LIN {X 0,Y 321.804,Z 530.514,A -85,B 0,C 180,E1 -15771.71,E2 -15771.71} C_VEL
LIN {X 0,Y 322.657,Z 517.307,A -85,B 0,C 180,E1 -15772.365,E2 -15772.365} C_VEL
LIN {X 0,Y 323.2,Z 504.38,A -85,B 0,C 180,E1 -15772.747,E2 -15772.747} C_VEL
LIN {X 0,Y 324.606,Z 436.447,A -85,B 0,C 180,E1 -15774.249,E2 -15774.249} C_VEL
LIN {X 0,Y 321.895,Z 423.016,A -85,B 0,C 180,E1 -15774.791,E2 -15774.791} C_VEL
LIN {X 0,Y 315.381,Z 406.695,A -85,B 0,C 180,E1 -15775.746,E2 -15775.746} C_VEL
LIN {X 0,Y 314.625,Z 404.517,A -85,B 0,C 180,E1 -15775.889,E2 -15775.889} C_VEL
LIN {X 0,Y 312.586,Z 395.049,A -85,B 0,C 180,E1 -15779.228,E2 -15779.228} C_VEL
LIN {X 0,Y 312.512,Z 395.055,A -85,B 0,C 180,E1 -15783.492,E2 -15783.492} C_VEL
LIN {X 0,Y 312.529,Z 395.054,A -85,B 0,C 180,E1 -15787.385,E2 -15787.385} C_VEL
LIN {X 0,Y 312.504,Z 395.058,A -85,B 0,C 180,E1 -15789.07,E2 -15789.07} C_VEL
LIN {X 0,Y 311.809,Z 395.146,A -85,B 0,C 180,E1 -15790.146,E2 -15790.146} C_VEL
LIN {X 0,Y 308.949,Z 395.503,A -85,B 0,C 180,E1 -15791.898,E2 -15791.898} C_VEL
LIN {X 0,Y 306.537,Z 395.806,A -85,B 0,C 180,E1 -15793.318,E2 -15793.318} C_VEL
LIN {X 0,Y 305.5,Z 395.932,A -85,B 0,C 180,E1 -15794.418,E2 -15794.418} C_VEL
LIN {X 0,Y 305.412,Z 395.941,A -85,B 0,C 180,E1 -15794.79,E2 -15794.79} C_VEL
LIN {X 0,Y 305.469,Z 395.935,A -85,B 0,C 180,E1 -15798.148,E2 -15798.148} C_VEL
LIN {X 0,Y 305.507,Z 395.922,A -85,B 0,C 180,E1 -15801.602,E2 -15801.602} C_VEL
LIN {X 0,Y 305.467,Z 395.933,A -85,B 0,C 180,E1 -15804.887,E2 -15804.887} C_VEL
LIN {X 0,Y 305.457,Z 395.938,A -85,B 0,C 180,E1 -15808.355,E2 -15808.355} C_VEL
LIN {X 0,Y 305.525,Z 395.924,A -85,B 0,C 180,E1 -15811.114,E2 -15811.114} C_VEL
LIN {X 0,Y 305.576,Z 395.922,A -85,B 0,C 180,E1 -15814.088,E2 -15814.088} C_VEL
LIN {X 0,Y 305.533,Z 395.926,A -85,B 0,C 180,E1 -15818.405,E2 -15818.405} C_VEL
LIN {X 0,Y 305.596,Z 395.913,A -85,B 0,C 180,E1 -15821.218,E2 -15821.218} C_VEL
LIN {X 0,Y 305.653,Z 395.908,A -85,B 0,C 180,E1 -15825.349,E2 -15825.349} C_VEL
LIN {X 0,Y 305.643,Z 395.911,A -85,B 0,C 180,E1 -15829.4,E2 -15829.4} C_VEL
LIN {X 0,Y 305.818,Z 395.887,A -85,B 0,C 180,E1 -15832.074,E2 -15832.074} C_VEL
LIN {X 0,Y 305.694,Z 395.904,A -85,B 0,C 180,E1 -15834.723,E2 -15834.723} C_VEL
LIN {X 0,Y 305.96,Z 395.866,A -85,B 0,C 180,E1 -15838.684,E2 -15838.684} C_VEL
LIN {X 0,Y 305.96,Z 395.871,A -85,B 0,C 180,E1 -15841.316,E2 -15841.316} C_VEL
LIN {X 0,Y 305.69,Z 395.903,A -85,B 0,C 180,E1 -15845.276,E2 -15845.276} C_VEL
LIN {X 0,Y 305.777,Z 395.897,A -85,B 0,C 180,E1 -15847.927,E2 -15847.927} C_VEL
LIN {X 0,Y 305.61,Z 395.915,A -85,B 0,C 180,E1 -15851.945,E2 -15851.945} C_VEL
LIN {X 0,Y 305.642,Z 395.911,A -85,B 0,C 180,E1 -15855.035,E2 -15855.035} C_VEL
LIN {X 0,Y 305.581,Z 395.922,A -85,B 0,C 180,E1 -15859.445,E2 -15859.445} C_VEL
LIN {X 0,Y 305.495,Z 395.927,A -85,B 0,C 180,E1 -15863.041,E2 -15863.041} C_VEL
LIN {X 0,Y 305.535,Z 395.924,A -85,B 0,C 180,E1 -15866.221,E2 -15866.221} C_VEL
LIN {X 0,Y 305.492,Z 395.931,A -85,B 0,C 180,E1 -15869.047,E2 -15869.047} C_VEL
LIN {X 0,Y 305.445,Z 395.935,A -85,B 0,C 180,E1 -15871.952,E2 -15871.952} C_VEL
LIN {X 0,Y 305.466,Z 395.935,A -85,B 0,C 180,E1 -15875.113,E2 -15875.113} C_VEL
LIN {X 0,Y 305.443,Z 395.935,A -85,B 0,C 180,E1 -15878.526,E2 -15878.526} C_VEL
LIN {X 0,Y 305.462,Z 395.934,A -85,B 0,C 180,E1 -15882.586,E2 -15882.586} C_VEL
LIN {X 0,Y 305.445,Z 395.936,A -85,B 0,C 180,E1 -15886.348,E2 -15886.348} C_VEL
LIN {X 0,Y 305.461,Z 395.934,A -85,B 0,C 180,E1 -15889.892,E2 -15889.892} C_VEL
LIN {X 0,Y 305.484,Z 395.933,A -85,B 0,C 180,E1 -15893.631,E2 -15893.631} C_VEL
LIN {X 0,Y 305.546,Z 396.115,A -85,B 0,C 180,E1 -15896.789,E2 -15896.789} C_VEL
LIN {X 0,Y 308.175,Z 407.817,A -85,B 0,C 180,E1 -15900.722,E2 -15900.722} C_VEL
LIN {X 0,Y 310.062,Z 417.52,A -85,B 0,C 180,E1 -15903.763,E2 -15903.763} C_VEL
LIN {X 0,Y 311.791,Z 423.086,A -85,B 0,C 180,E1 -15904.058,E2 -15904.058} C_VEL
LIN {X 0,Y 316.195,Z 447.46,A -85,B 0,C 180,E1 -15905.042,E2 -15905.042} C_VEL
LIN {X 0,Y 317.783,Z 458.385,A -85,B 0,C 180,E1 -15905.441,E2 -15905.441} C_VEL
LIN {X 0,Y 316.113,Z 525.615,A -85,B 0,C 180,E1 -15906.973,E2 -15906.973} C_VEL
LIN {X 0,Y 315.252,Z 538.795,A -85,B 0,C 180,E1 -15907.513,E2 -15907.513} C_VEL
LIN {X 0,Y 314.171,Z 550.908,A -85,B 0,C 180,E1 -15908.253,E2 -15908.253} C_VEL
LIN {X 0,Y 312.715,Z 563.132,A -85,B 0,C 180,E1 -15909.269,E2 -15909.269} C_VEL
LIN {X 0,Y 311.16,Z 574.706,A -85,B 0,C 180,E1 -15910.54,E2 -15910.54} C_VEL
LIN {X 0,Y 309.557,Z 585.128,A -85,B 0,C 180,E1 -15911.981,E2 -15911.981} C_VEL
LIN {X 0,Y 308.213,Z 594.648,A -85,B 0,C 180,E1 -15913.638,E2 -15913.638} C_VEL
LIN {X 0,Y 306.919,Z 602.895,A -85,B 0,C 180,E1 -15915.411,E2 -15915.411} C_VEL
LIN {X 0,Y 305.617,Z 610.319,A -85,B 0,C 180,E1 -15917.381,E2 -15917.381} C_VEL
LIN {X 0,Y 304.721,Z 616.285,A -85,B 0,C 180,E1 -15919.367,E2 -15919.367} C_VEL
LIN {X 0,Y 304.15,Z 621.001,A -85,B 0,C 180,E1 -15921.361,E2 -15921.361} C_VEL
LIN {X 0,Y 303.741,Z 624.604,A -85,B 0,C 180,E1 -15923.356,E2 -15923.356} C_VEL
LIN {X 0,Y 303.618,Z 626.463,A -85,B 0,C 180,E1 -15924.687,E2 -15924.687} C_VEL
LIN {X 0,Y 303.589,Z 627.858,A -85,B 0,C 180,E1 -15926.017,E2 -15926.017} C_VEL
LIN {X 0,Y 303.598,Z 628.855,A -85,B 0,C 180,E1 -15927.346,E2 -15927.346} C_VEL
LIN {X 0,Y 303.556,Z 629.461,A -85,B 0,C 180,E1 -15928.673,E2 -15928.673} C_VEL
LIN {X 0,Y 303.565,Z 629.674,A -85,B 0,C 180,E1 -15930,E2 -15930} C_VEL
LIN {X 0,Y 303.556,Z 629.454,A -85,B 0,C 180,E1 -15931.326,E2 -15931.326} C_VEL
LIN {X 0,Y 303.598,Z 628.844,A -85,B 0,C 180,E1 -15932.653,E2 -15932.653} C_VEL
LIN {X 0,Y 303.589,Z 627.844,A -85,B 0,C 180,E1 -15933.982,E2 -15933.982} C_VEL
LIN {X 0,Y 303.618,Z 626.155,A -85,B 0,C 180,E1 -15935.53,E2 -15935.53} C_VEL
LIN {X 0,Y 303.993,Z 622.272,A -85,B 0,C 180,E1 -15937.973,E2 -15937.973} C_VEL
LIN {X 0,Y 304.49,Z 617.927,A -85,B 0,C 180,E1 -15939.968,E2 -15939.968} C_VEL
LIN {X 0,Y 305.24,Z 612.394,A -85,B 0,C 180,E1 -15941.959,E2 -15941.959} C_VEL
LIN {X 0,Y 306.422,Z 605.493,A -85,B 0,C 180,E1 -15943.935,E2 -15943.935} C_VEL
LIN {X 0,Y 307.55,Z 598.445,A -85,B 0,C 180,E1 -15945.575,E2 -15945.575} C_VEL
LIN {X 0,Y 308.841,Z 589.95,A -85,B 0,C 180,E1 -15947.207,E2 -15947.207} C_VEL
LIN {X 0,Y 310.402,Z 579.455,A -85,B 0,C 180,E1 -15948.823,E2 -15948.823} C_VEL
LIN {X 0,Y 312.114,Z 567.645,A -85,B 0,C 180,E1 -15950.255,E2 -15950.255} C_VEL
LIN {X 0,Y 313.542,Z 555.751,A -85,B 0,C 180,E1 -15951.361,E2 -15951.361} C_VEL
LIN {X 0,Y 314.779,Z 543.373,A -85,B 0,C 180,E1 -15952.22,E2 -15952.22} C_VEL
LIN {X 0,Y 315.807,Z 530.636,A -85,B 0,C 180,E1 -15952.833,E2 -15952.833} C_VEL
LIN {X 0,Y 316.361,Z 517.195,A -85,B 0,C 180,E1 -15953.223,E2 -15953.223} C_VEL
LIN {X 0,Y 317.613,Z 456.986,A -85,B 0,C 180,E1 -15954.583,E2 -15954.583} C_VEL
LIN {X 0,Y 313.2,Z 430.545,A -85,B 0,C 180,E1 -15955.606,E2 -15955.606} C_VEL
LIN {X 0,Y 311.031,Z 420.234,A -85,B 0,C 180,E1 -15956.055,E2 -15956.055} C_VEL
LIN {X 0,Y 309.994,Z 417.236,A -85,B 0,C 180,E1 -15956.25,E2 -15956.25} C_VEL
LIN {X 0,Y 308.239,Z 408.025,A -85,B 0,C 180,E1 -15959.181,E2 -15959.181} C_VEL
LIN {X 0,Y 305.506,Z 395.931,A -85,B 0,C 180,E1 -15963.265,E2 -15963.265} C_VEL
LIN {X 0,Y 305.476,Z 395.934,A -85,B 0,C 180,E1 -15966.739,E2 -15966.739} C_VEL
LIN {X 0,Y 305.455,Z 395.936,A -85,B 0,C 180,E1 -15970.6,E2 -15970.6} C_VEL
LIN {X 0,Y 305.42,Z 395.939,A -85,B 0,C 180,E1 -15974.493,E2 -15974.493} C_VEL
LIN {X 0,Y 305.443,Z 395.935,A -85,B 0,C 180,E1 -15978.143,E2 -15978.143} C_VEL
LIN {X 0,Y 305.468,Z 395.93,A -85,B 0,C 180,E1 -15981.596,E2 -15981.596} C_VEL
LIN {X 0,Y 305.464,Z 395.934,A -85,B 0,C 180,E1 -15984.887,E2 -15984.887} C_VEL
LIN {X 0,Y 305.451,Z 395.936,A -85,B 0,C 180,E1 -15988.356,E2 -15988.356} C_VEL
LIN {X 0,Y 305.514,Z 395.927,A -85,B 0,C 180,E1 -15991.113,E2 -15991.113} C_VEL
LIN {X 0,Y 305.572,Z 395.92,A -85,B 0,C 180,E1 -15994.088,E2 -15994.088} C_VEL
LIN {X 0,Y 305.528,Z 395.928,A -85,B 0,C 180,E1 -15998.405,E2 -15998.405} C_VEL
LIN {X 0,Y 305.592,Z 395.916,A -85,B 0,C 180,E1 -16001.218,E2 -16001.218} C_VEL
LIN {X 0,Y 305.651,Z 395.906,A -85,B 0,C 180,E1 -16005.349,E2 -16005.349} C_VEL
LIN {X 0,Y 305.639,Z 395.909,A -85,B 0,C 180,E1 -16009.4,E2 -16009.4} C_VEL
LIN {X 0,Y 305.774,Z 395.896,A -85,B 0,C 180,E1 -16012.073,E2 -16012.073} C_VEL
LIN {X 0,Y 305.686,Z 395.904,A -85,B 0,C 180,E1 -16014.723,E2 -16014.723} C_VEL
LIN {X 0,Y 305.958,Z 395.872,A -85,B 0,C 180,E1 -16018.684,E2 -16018.684} C_VEL
LIN {X 0,Y 305.96,Z 395.867,A -85,B 0,C 180,E1 -16021.316,E2 -16021.316} C_VEL
LIN {X 0,Y 305.855,Z 395.883,A -85,B 0,C 180,E1 -16026.597,E2 -16026.597} C_VEL
LIN {X 0,Y 305.737,Z 395.899,A -85,B 0,C 180,E1 -16029.26,E2 -16029.26} C_VEL
LIN {X 0,Y 305.591,Z 395.916,A -85,B 0,C 180,E1 -16033.296,E2 -16033.296} C_VEL
LIN {X 0,Y 305.596,Z 395.918,A -85,B 0,C 180,E1 -16036.02,E2 -16036.02} C_VEL
LIN {X 0,Y 305.583,Z 395.919,A -85,B 0,C 180,E1 -16039.447,E2 -16039.447} C_VEL
LIN {X 0,Y 305.493,Z 395.928,A -85,B 0,C 180,E1 -16043.042,E2 -16043.042} C_VEL
LIN {X 0,Y 305.549,Z 395.922,A -85,B 0,C 180,E1 -16046.227,E2 -16046.227} C_VEL
LIN {X 0,Y 305.497,Z 395.929,A -85,B 0,C 180,E1 -16049.05,E2 -16049.05} C_VEL
LIN {X 0,Y 305.447,Z 395.938,A -85,B 0,C 180,E1 -16051.952,E2 -16051.952} C_VEL
LIN {X 0,Y 305.465,Z 395.932,A -85,B 0,C 180,E1 -16055.113,E2 -16055.113} C_VEL
LIN {X 0,Y 305.479,Z 395.93,A -85,B 0,C 180,E1 -16058.536,E2 -16058.536} C_VEL
LIN {X 0,Y 305.476,Z 395.931,A -85,B 0,C 180,E1 -16062.59,E2 -16062.59} C_VEL
LIN {X 0,Y 305.456,Z 395.936,A -85,B 0,C 180,E1 -16067.414,E2 -16067.414} C_VEL
LIN {X 0,Y 305.478,Z 395.934,A -85,B 0,C 180,E1 -16071.598,E2 -16071.598} C_VEL
LIN {X 0,Y 305.464,Z 395.935,A -85,B 0,C 180,E1 -16074.887,E2 -16074.887} C_VEL
LIN {X 0,Y 305.454,Z 395.937,A -85,B 0,C 180,E1 -16078.355,E2 -16078.355} C_VEL
LIN {X 0,Y 305.519,Z 395.981,A -85,B 0,C 180,E1 -16080.42,E2 -16080.42} C_VEL
LIN {X 0,Y 307.484,Z 404.768,A -85,B 0,C 180,E1 -16083.603,E2 -16083.603} C_VEL
LIN {X 0,Y 315.927,Z 426.072,A -85,B 0,C 180,E1 -16084.895,E2 -16084.895} C_VEL
LIN {X 0,Y 318.22,Z 437.996,A -85,B 0,C 180,E1 -16085.381,E2 -16085.381} C_VEL
LIN {X 0,Y 316.423,Z 511.235,A -85,B 0,C 180,E1 -16087.041,E2 -16087.041} C_VEL
LIN {X 0,Y 315.6,Z 524.625,A -85,B 0,C 180,E1 -16087.583,E2 -16087.583} C_VEL
LIN {X 0,Y 314.558,Z 537.389,A -85,B 0,C 180,E1 -16088.368,E2 -16088.368} C_VEL
LIN {X 0,Y 313.347,Z 548.722,A -85,B 0,C 180,E1 -16089.314,E2 -16089.314} C_VEL
LIN {X 0,Y 311.903,Z 560.369,A -85,B 0,C 180,E1 -16090.588,E2 -16090.588} C_VEL
LIN {X 0,Y 310.383,Z 571.362,A -85,B 0,C 180,E1 -16092.117,E2 -16092.117} C_VEL
LIN {X 0,Y 308.925,Z 581.06,A -85,B 0,C 180,E1 -16093.818,E2 -16093.818} C_VEL
LIN {X 0,Y 307.357,Z 589.977,A -85,B 0,C 180,E1 -16095.771,E2 -16095.771} C_VEL
LIN {X 0,Y 306.173,Z 597.152,A -85,B 0,C 180,E1 -16097.741,E2 -16097.741} C_VEL
LIN {X 0,Y 305.366,Z 601.99,A -85,B 0,C 180,E1 -16099.39,E2 -16099.39} C_VEL
LIN {X 0,Y 304.611,Z 606.691,A -85,B 0,C 180,E1 -16101.375,E2 -16101.375} C_VEL
LIN {X 0,Y 304.105,Z 610.649,A -85,B 0,C 180,E1 -16103.593,E2 -16103.593} C_VEL
LIN {X 0,Y 303.82,Z 613.541,A -85,B 0,C 180,E1 -16106.021,E2 -16106.021} C_VEL
LIN {X 0,Y 303.598,Z 615.148,A -85,B 0,C 180,E1 -16108.674,E2 -16108.674} C_VEL
LIN {X 0,Y 303.571,Z 615.38,A -85,B 0,C 180,E1 -16110,E2 -16110} C_VEL
LIN {X 0,Y 303.598,Z 615.187,A -85,B 0,C 180,E1 -16111.327,E2 -16111.327} C_VEL
LIN {X 0,Y 303.817,Z 613.631,A -85,B 0,C 180,E1 -16113.98,E2 -16113.98} C_VEL
LIN {X 0,Y 304.071,Z 610.898,A -85,B 0,C 180,E1 -16116.35,E2 -16116.35} C_VEL
LIN {X 0,Y 304.609,Z 606.928,A -85,B 0,C 180,E1 -16118.625,E2 -16118.625} C_VEL
LIN {X 0,Y 305.318,Z 602.291,A -85,B 0,C 180,E1 -16120.612,E2 -16120.612} C_VEL
LIN {X 0,Y 306.51,Z 595.298,A -85,B 0,C 180,E1 -16122.918,E2 -16122.918} C_VEL
LIN {X 0,Y 307.787,Z 587.719,A -85,B 0,C 180,E1 -16124.885,E2 -16124.885} C_VEL
LIN {X 0,Y 309.433,Z 578.177,A -85,B 0,C 180,E1 -16126.833,E2 -16126.833} C_VEL
LIN {X 0,Y 310.835,Z 568.331,A -85,B 0,C 180,E1 -16128.454,E2 -16128.454} C_VEL
LIN {X 0,Y 312.169,Z 558.637,A -85,B 0,C 180,E1 -16129.737,E2 -16129.737} C_VEL
LIN {X 0,Y 313.521,Z 548.137,A -85,B 0,C 180,E1 -16130.847,E2 -16130.847} C_VEL
LIN {X 0,Y 314.84,Z 535.491,A -85,B 0,C 180,E1 -16131.871,E2 -16131.871} C_VEL
LIN {X 0,Y 315.792,Z 522.821,A -85,B 0,C 180,E1 -16132.619,E2 -16132.619} C_VEL
LIN {X 0,Y 316.469,Z 510.728,A -85,B 0,C 180,E1 -16133.086,E2 -16133.086} C_VEL
LIN {X 0,Y 318.156,Z 437.661,A -85,B 0,C 180,E1 -16134.747,E2 -16134.747} C_VEL
LIN {X 0,Y 315.68,Z 425.321,A -85,B 0,C 180,E1 -16135.26,E2 -16135.26} C_VEL
LIN {X 0,Y 308.519,Z 407.482,A -85,B 0,C 180,E1 -16136.346,E2 -16136.346} C_VEL
LIN {X 0,Y 307.462,Z 404.709,A -85,B 0,C 180,E1 -16136.533,E2 -16136.533} C_VEL
LIN {X 0,Y 305.524,Z 395.929,A -85,B 0,C 180,E1 -16139.776,E2 -16139.776} C_VEL
LIN {X 0,Y 305.468,Z 395.934,A -85,B 0,C 180,E1 -16144.079,E2 -16144.079} C_VEL
LIN {X 0,Y 305.478,Z 395.932,A -85,B 0,C 180,E1 -16146.74,E2 -16146.74} C_VEL
LIN {X 0,Y 305.458,Z 395.937,A -85,B 0,C 180,E1 -16150.6,E2 -16150.6} C_VEL
LIN {X 0,Y 305.422,Z 395.942,A -85,B 0,C 180,E1 -16154.493,E2 -16154.493} C_VEL
LIN {X 0,Y 305.412,Z 395.941,A -85,B 0,C 180,E1 -16154.79,E2 -16154.79} C_VEL
LIN {X 0,Y 304.74,Z 396.024,A -85,B 0,C 180,E1 -16155.891,E2 -16155.891} C_VEL
LIN {X 0,Y 301.904,Z 396.377,A -85,B 0,C 180,E1 -16157.684,E2 -16157.684} C_VEL
LIN {X 0,Y 299.511,Z 396.67,A -85,B 0,C 180,E1 -16159.138,E2 -16159.138} C_VEL
LIN {X 0,Y 298.494,Z 396.795,A -85,B 0,C 180,E1 -16160.264,E2 -16160.264} C_VEL
LIN {X 0,Y 298.417,Z 396.804,A -85,B 0,C 180,E1 -16160.645,E2 -16160.645} C_VEL
LIN {X 0,Y 298.436,Z 396.809,A -85,B 0,C 180,E1 -16163.932,E2 -16163.932} C_VEL
LIN {X 0,Y 298.4,Z 396.815,A -85,B 0,C 180,E1 -16167.983,E2 -16167.983} C_VEL
LIN {X 0,Y 298.468,Z 396.805,A -85,B 0,C 180,E1 -16171.905,E2 -16171.905} C_VEL
LIN {X 0,Y 298.49,Z 396.798,A -85,B 0,C 180,E1 -16174.924,E2 -16174.924} C_VEL
LIN {X 0,Y 298.469,Z 396.803,A -85,B 0,C 180,E1 -16179.317,E2 -16179.317} C_VEL
LIN {X 0,Y 298.543,Z 396.797,A -85,B 0,C 180,E1 -16182.18,E2 -16182.18} C_VEL
LIN {X 0,Y 298.598,Z 396.787,A -85,B 0,C 180,E1 -16184.995,E2 -16184.995} C_VEL
LIN {X 0,Y 298.598,Z 396.788,A -85,B 0,C 180,E1 -16189.147,E2 -16189.147} C_VEL
LIN {X 0,Y 298.763,Z 396.767,A -85,B 0,C 180,E1 -16191.886,E2 -16191.886} C_VEL
LIN {X 0,Y 298.665,Z 396.78,A -85,B 0,C 180,E1 -16194.599,E2 -16194.599} C_VEL
LIN {X 0,Y 298.927,Z 396.742,A -85,B 0,C 180,E1 -16198.653,E2 -16198.653} C_VEL
LIN {X 0,Y 298.927,Z 396.747,A -85,B 0,C 180,E1 -16201.347,E2 -16201.347} C_VEL
LIN {X 0,Y 298.782,Z 396.763,A -85,B 0,C 180,E1 -16206.754,E2 -16206.754} C_VEL
LIN {X 0,Y 298.636,Z 396.787,A -85,B 0,C 180,E1 -16209.482,E2 -16209.482} C_VEL
LIN {X 0,Y 298.558,Z 396.796,A -85,B 0,C 180,E1 -16213.615,E2 -16213.615} C_VEL
LIN {X 0,Y 298.553,Z 396.791,A -85,B 0,C 180,E1 -16216.408,E2 -16216.408} C_VEL
LIN {X 0,Y 298.516,Z 396.802,A -85,B 0,C 180,E1 -16219.655,E2 -16219.655} C_VEL
LIN {X 0,Y 298.461,Z 396.808,A -85,B 0,C 180,E1 -16223.597,E2 -16223.597} C_VEL
LIN {X 0,Y 298.49,Z 396.801,A -85,B 0,C 180,E1 -16226.574,E2 -16226.574} C_VEL
LIN {X 0,Y 298.42,Z 396.812,A -85,B 0,C 180,E1 -16229.641,E2 -16229.641} C_VEL
LIN {X 0,Y 298.398,Z 396.813,A -85,B 0,C 180,E1 -16232.8,E2 -16232.8} C_VEL
LIN {X 0,Y 298.447,Z 396.808,A -85,B 0,C 180,E1 -16236.807,E2 -16236.807} C_VEL
LIN {X 0,Y 298.391,Z 396.818,A -85,B 0,C 180,E1 -16241.088,E2 -16241.088} C_VEL
LIN {X 0,Y 298.391,Z 396.818,A -85,B 0,C 180,E1 -16245.041,E2 -16245.041} C_VEL
LIN {X 0,Y 298.391,Z 396.818,A -85,B 0,C 180,E1 -16248.912,E2 -16248.912} C_VEL
LIN {X 0,Y 298.449,Z 396.81,A -85,B 0,C 180,E1 -16253.192,E2 -16253.192} C_VEL
LIN {X 0,Y 298.451,Z 396.866,A -85,B 0,C 180,E1 -16256.197,E2 -16256.197} C_VEL
LIN {X 0,Y 300.988,Z 407.974,A -85,B 0,C 180,E1 -16260.058,E2 -16260.058} C_VEL
LIN {X 0,Y 302.821,Z 417.308,A -85,B 0,C 180,E1 -16263.085,E2 -16263.085} C_VEL
LIN {X 0,Y 305.502,Z 424.753,A -85,B 0,C 180,E1 -16263.53,E2 -16263.53} C_VEL
LIN {X 0,Y 309.917,Z 449.444,A -85,B 0,C 180,E1 -16264.554,E2 -16264.554} C_VEL
LIN {X 0,Y 311.305,Z 459.53,A -85,B 0,C 180,E1 -16264.927,E2 -16264.927} C_VEL
LIN {X 0,Y 309.595,Z 525.461,A -85,B 0,C 180,E1 -16266.46,E2 -16266.46} C_VEL
LIN {X 0,Y 308.704,Z 538.637,A -85,B 0,C 180,E1 -16267.009,E2 -16267.009} C_VEL
LIN {X 0,Y 307.593,Z 550.747,A -85,B 0,C 180,E1 -16267.763,E2 -16267.763} C_VEL
LIN {X 0,Y 306.089,Z 562.97,A -85,B 0,C 180,E1 -16268.799,E2 -16268.799} C_VEL
LIN {X 0,Y 304.483,Z 574.543,A -85,B 0,C 180,E1 -16270.095,E2 -16270.095} C_VEL
LIN {X 0,Y 302.773,Z 584.963,A -85,B 0,C 180,E1 -16271.562,E2 -16271.562} C_VEL
LIN {X 0,Y 301.516,Z 593.488,A -85,B 0,C 180,E1 -16273.06,E2 -16273.06} C_VEL
LIN {X 0,Y 300.281,Z 601.354,A -85,B 0,C 180,E1 -16274.733,E2 -16274.733} C_VEL
LIN {X 0,Y 298.857,Z 609.032,A -85,B 0,C 180,E1 -16276.745,E2 -16276.745} C_VEL
LIN {X 0,Y 297.727,Z 616.119,A -85,B 0,C 180,E1 -16279.114,E2 -16279.114} C_VEL
LIN {X 0,Y 297.092,Z 620.834,A -85,B 0,C 180,E1 -16281.155,E2 -16281.155} C_VEL
LIN {X 0,Y 296.688,Z 624.438,A -85,B 0,C 180,E1 -16283.198,E2 -16283.198} C_VEL
LIN {X 0,Y 296.532,Z 626.296,A -85,B 0,C 180,E1 -16284.56,E2 -16284.56} C_VEL
LIN {X 0,Y 296.49,Z 627.691,A -85,B 0,C 180,E1 -16285.922,E2 -16285.922} C_VEL
LIN {X 0,Y 296.523,Z 628.688,A -85,B 0,C 180,E1 -16287.283,E2 -16287.283} C_VEL
LIN {X 0,Y 296.476,Z 629.294,A -85,B 0,C 180,E1 -16288.641,E2 -16288.641} C_VEL
LIN {X 0,Y 296.482,Z 629.508,A -85,B 0,C 180,E1 -16290,E2 -16290} C_VEL
LIN {X 0,Y 296.476,Z 629.287,A -85,B 0,C 180,E1 -16291.358,E2 -16291.358} C_VEL
LIN {X 0,Y 296.523,Z 628.677,A -85,B 0,C 180,E1 -16292.717,E2 -16292.717} C_VEL
LIN {X 0,Y 296.49,Z 627.677,A -85,B 0,C 180,E1 -16294.078,E2 -16294.078} C_VEL
LIN {X 0,Y 296.546,Z 626.189,A -85,B 0,C 180,E1 -16295.508,E2 -16295.508} C_VEL
LIN {X 0,Y 296.796,Z 623.333,A -85,B 0,C 180,E1 -16297.483,E2 -16297.483} C_VEL
LIN {X 0,Y 297.274,Z 619.354,A -85,B 0,C 180,E1 -16299.526,E2 -16299.526} C_VEL
LIN {X 0,Y 298.128,Z 613.237,A -85,B 0,C 180,E1 -16301.904,E2 -16301.904} C_VEL
LIN {X 0,Y 299.301,Z 606.56,A -85,B 0,C 180,E1 -16303.927,E2 -16303.927} C_VEL
LIN {X 0,Y 300.683,Z 598.275,A -85,B 0,C 180,E1 -16305.94,E2 -16305.94} C_VEL
LIN {X 0,Y 302.043,Z 589.78,A -85,B 0,C 180,E1 -16307.607,E2 -16307.607} C_VEL
LIN {X 0,Y 303.666,Z 579.284,A -85,B 0,C 180,E1 -16309.256,E2 -16309.256} C_VEL
LIN {X 0,Y 305.454,Z 567.473,A -85,B 0,C 180,E1 -16310.717,E2 -16310.717} C_VEL
LIN {X 0,Y 306.952,Z 555.579,A -85,B 0,C 180,E1 -16311.843,E2 -16311.843} C_VEL
LIN {X 0,Y 308.219,Z 543.198,A -85,B 0,C 180,E1 -16312.719,E2 -16312.719} C_VEL
LIN {X 0,Y 309.285,Z 530.458,A -85,B 0,C 180,E1 -16313.343,E2 -16313.343} C_VEL
LIN {X 0,Y 309.851,Z 517.007,A -85,B 0,C 180,E1 -16313.741,E2 -16313.741} C_VEL
LIN {X 0,Y 311.196,Z 458.096,A -85,B 0,C 180,E1 -16315.093,E2 -16315.093} C_VEL
LIN {X 0,Y 306.801,Z 431.766,A -85,B 0,C 180,E1 -16316.144,E2 -16316.144} C_VEL
LIN {X 0,Y 304.983,Z 422.969,A -85,B 0,C 180,E1 -16316.537,E2 -16316.537} C_VEL
LIN {X 0,Y 302.765,Z 417.024,A -85,B 0,C 180,E1 -16316.935,E2 -16316.935} C_VEL
LIN {X 0,Y 300.809,Z 407.187,A -85,B 0,C 180,E1 -16320.179,E2 -16320.179} C_VEL
LIN {X 0,Y 298.45,Z 396.81,A -85,B 0,C 180,E1 -16323.802,E2 -16323.802} C_VEL
LIN {X 0,Y 298.415,Z 396.812,A -85,B 0,C 180,E1 -16327.758,E2 -16327.758} C_VEL
LIN {X 0,Y 298.386,Z 396.816,A -85,B 0,C 180,E1 -16331.261,E2 -16331.261} C_VEL
LIN {X 0,Y 298.389,Z 396.818,A -85,B 0,C 180,E1 -16335.041,E2 -16335.041} C_VEL
LIN {X 0,Y 298.389,Z 396.815,A -85,B 0,C 180,E1 -16338.912,E2 -16338.912} C_VEL
LIN {X 0,Y 298.445,Z 396.808,A -85,B 0,C 180,E1 -16343.193,E2 -16343.193} C_VEL
LIN {X 0,Y 298.396,Z 396.814,A -85,B 0,C 180,E1 -16347.2,E2 -16347.2} C_VEL
LIN {X 0,Y 298.428,Z 396.813,A -85,B 0,C 180,E1 -16350.616,E2 -16350.616} C_VEL
LIN {X 0,Y 298.479,Z 396.803,A -85,B 0,C 180,E1 -16353.476,E2 -16353.476} C_VEL
LIN {X 0,Y 298.437,Z 396.81,A -85,B 0,C 180,E1 -16356.697,E2 -16356.697} C_VEL
LIN {X 0,Y 298.541,Z 396.796,A -85,B 0,C 180,E1 -16360.757,E2 -16360.757} C_VEL
LIN {X 0,Y 298.595,Z 396.786,A -85,B 0,C 180,E1 -16364.995,E2 -16364.995} C_VEL
LIN {X 0,Y 298.595,Z 396.787,A -85,B 0,C 180,E1 -16369.147,E2 -16369.147} C_VEL
LIN {X 0,Y 298.72,Z 396.773,A -85,B 0,C 180,E1 -16371.885,E2 -16371.885} C_VEL
LIN {X 0,Y 298.657,Z 396.78,A -85,B 0,C 180,E1 -16374.599,E2 -16374.599} C_VEL
LIN {X 0,Y 298.924,Z 396.749,A -85,B 0,C 180,E1 -16378.653,E2 -16378.653} C_VEL
LIN {X 0,Y 298.926,Z 396.743,A -85,B 0,C 180,E1 -16381.347,E2 -16381.347} C_VEL
LIN {X 0,Y 298.8,Z 396.761,A -85,B 0,C 180,E1 -16386.754,E2 -16386.754} C_VEL
LIN {X 0,Y 298.682,Z 396.778,A -85,B 0,C 180,E1 -16389.481,E2 -16389.481} C_VEL
LIN {X 0,Y 298.554,Z 396.794,A -85,B 0,C 180,E1 -16393.615,E2 -16393.615} C_VEL
LIN {X 0,Y 298.551,Z 396.792,A -85,B 0,C 180,E1 -16396.409,E2 -16396.409} C_VEL
LIN {X 0,Y 298.518,Z 396.801,A -85,B 0,C 180,E1 -16399.657,E2 -16399.657} C_VEL
LIN {X 0,Y 298.459,Z 396.807,A -85,B 0,C 180,E1 -16403.598,E2 -16403.598} C_VEL
LIN {X 0,Y 298.491,Z 396.8,A -85,B 0,C 180,E1 -16406.574,E2 -16406.574} C_VEL
LIN {X 0,Y 298.422,Z 396.813,A -85,B 0,C 180,E1 -16409.641,E2 -16409.641} C_VEL
LIN {X 0,Y 298.398,Z 396.813,A -85,B 0,C 180,E1 -16412.8,E2 -16412.8} C_VEL
LIN {X 0,Y 298.467,Z 396.804,A -85,B 0,C 180,E1 -16416.813,E2 -16416.813} C_VEL
LIN {X 0,Y 298.415,Z 396.811,A -85,B 0,C 180,E1 -16421.094,E2 -16421.094} C_VEL
LIN {X 0,Y 298.355,Z 396.819,A -85,B 0,C 180,E1 -16425.035,E2 -16425.035} C_VEL
LIN {X 0,Y 298.386,Z 396.816,A -85,B 0,C 180,E1 -16428.739,E2 -16428.739} C_VEL
LIN {X 0,Y 298.416,Z 396.812,A -85,B 0,C 180,E1 -16432.242,E2 -16432.242} C_VEL
LIN {X 0,Y 298.41,Z 396.814,A -85,B 0,C 180,E1 -16435.581,E2 -16435.581} C_VEL
LIN {X 0,Y 298.468,Z 396.936,A -85,B 0,C 180,E1 -16439.927,E2 -16439.927} C_VEL
LIN {X 0,Y 300.277,Z 404.892,A -85,B 0,C 180,E1 -16442.896,E2 -16442.896} C_VEL
LIN {X 0,Y 308.044,Z 423.883,A -85,B 0,C 180,E1 -16444.144,E2 -16444.144} C_VEL
LIN {X 0,Y 310.011,Z 429.691,A -85,B 0,C 180,E1 -16444.468,E2 -16444.468} C_VEL
LIN {X 0,Y 311.75,Z 439.041,A -85,B 0,C 180,E1 -16444.856,E2 -16444.856} C_VEL
LIN {X 0,Y 309.917,Z 511.419,A -85,B 0,C 180,E1 -16446.53,E2 -16446.53} C_VEL
LIN {X 0,Y 309.071,Z 524.802,A -85,B 0,C 180,E1 -16447.082,E2 -16447.082} C_VEL
LIN {X 0,Y 307.986,Z 537.563,A -85,B 0,C 180,E1 -16447.882,E2 -16447.882} C_VEL
LIN {X 0,Y 306.731,Z 548.894,A -85,B 0,C 180,E1 -16448.846,E2 -16448.846} C_VEL
LIN {X 0,Y 305.216,Z 560.54,A -85,B 0,C 180,E1 -16450.145,E2 -16450.145} C_VEL
LIN {X 0,Y 303.81,Z 570.356,A -85,B 0,C 180,E1 -16451.523,E2 -16451.523} C_VEL
LIN {X 0,Y 302.431,Z 579.537,A -85,B 0,C 180,E1 -16453.113,E2 -16453.113} C_VEL
LIN {X 0,Y 301.009,Z 587.409,A -85,B 0,C 180,E1 -16454.772,E2 -16454.772} C_VEL
LIN {X 0,Y 299.647,Z 595.099,A -85,B 0,C 180,E1 -16456.781,E2 -16456.781} C_VEL
LIN {X 0,Y 298.385,Z 602.159,A -85,B 0,C 180,E1 -16459.139,E2 -16459.139} C_VEL
LIN {X 0,Y 297.592,Z 606.86,A -85,B 0,C 180,E1 -16461.17,E2 -16461.17} C_VEL
LIN {X 0,Y 297.024,Z 611.062,A -85,B 0,C 180,E1 -16463.608,E2 -16463.608} C_VEL
LIN {X 0,Y 296.738,Z 613.709,A -85,B 0,C 180,E1 -16465.926,E2 -16465.926} C_VEL
LIN {X 0,Y 296.61,Z 614.703,A -85,B 0,C 180,E1 -16467.284,E2 -16467.284} C_VEL
LIN {X 0,Y 296.488,Z 615.546,A -85,B 0,C 180,E1 -16470,E2 -16470} C_VEL
LIN {X 0,Y 296.518,Z 615.354,A -85,B 0,C 180,E1 -16471.358,E2 -16471.358} C_VEL
LIN {X 0,Y 296.609,Z 614.767,A -85,B 0,C 180,E1 -16472.716,E2 -16472.716} C_VEL
LIN {X 0,Y 296.736,Z 613.798,A -85,B 0,C 180,E1 -16474.075,E2 -16474.075} C_VEL
LIN {X 0,Y 296.997,Z 611.27,A -85,B 0,C 180,E1 -16476.345,E2 -16476.345} C_VEL
LIN {X 0,Y 297.59,Z 607.094,A -85,B 0,C 180,E1 -16478.831,E2 -16478.831} C_VEL
LIN {X 0,Y 298.341,Z 602.456,A -85,B 0,C 180,E1 -16480.863,E2 -16480.863} C_VEL
LIN {X 0,Y 299.557,Z 595.464,A -85,B 0,C 180,E1 -16483.224,E2 -16483.224} C_VEL
LIN {X 0,Y 300.94,Z 587.884,A -85,B 0,C 180,E1 -16485.232,E2 -16485.232} C_VEL
LIN {X 0,Y 302.638,Z 578.341,A -85,B 0,C 180,E1 -16487.223,E2 -16487.223} C_VEL
LIN {X 0,Y 304.094,Z 568.494,A -85,B 0,C 180,E1 -16488.879,E2 -16488.879} C_VEL
LIN {X 0,Y 305.506,Z 558.799,A -85,B 0,C 180,E1 -16490.186,E2 -16490.186} C_VEL
LIN {X 0,Y 306.91,Z 548.298,A -85,B 0,C 180,E1 -16491.317,E2 -16491.317} C_VEL
LIN {X 0,Y 308.255,Z 535.65,A -85,B 0,C 180,E1 -16492.363,E2 -16492.363} C_VEL
LIN {X 0,Y 309.267,Z 522.977,A -85,B 0,C 180,E1 -16493.124,E2 -16493.124} C_VEL
LIN {X 0,Y 309.969,Z 510.875,A -85,B 0,C 180,E1 -16493.599,E2 -16493.599} C_VEL
LIN {X 0,Y 311.742,Z 438.654,A -85,B 0,C 180,E1 -16495.27,E2 -16495.27} C_VEL
LIN {X 0,Y 309.528,Z 427.798,A -85,B 0,C 180,E1 -16495.739,E2 -16495.739} C_VEL
LIN {X 0,Y 302.552,Z 410.393,A -85,B 0,C 180,E1 -16496.835,E2 -16496.835} C_VEL
LIN {X 0,Y 300.286,Z 404.93,A -85,B 0,C 180,E1 -16497.206,E2 -16497.206} C_VEL
LIN {X 0,Y 298.451,Z 396.81,A -85,B 0,C 180,E1 -16500.32,E2 -16500.32} C_VEL
LIN {X 0,Y 298.431,Z 396.814,A -85,B 0,C 180,E1 -16504.488,E2 -16504.488} C_VEL
LIN {X 0,Y 298.417,Z 396.812,A -85,B 0,C 180,E1 -16507.758,E2 -16507.758} C_VEL
LIN {X 0,Y 298.388,Z 396.815,A -85,B 0,C 180,E1 -16511.262,E2 -16511.262} C_VEL
LIN {X 0,Y 298.391,Z 396.814,A -85,B 0,C 180,E1 -16515.042,E2 -16515.042} C_VEL
LIN {X 0,Y 298.417,Z 396.809,A -85,B 0,C 180,E1 -16518.744,E2 -16518.744} C_VEL
LIN {X 0,Y 298.417,Z 396.804,A -85,B 0,C 180,E1 -16520.645,E2 -16520.645} C_VEL
LIN {X 0,Y 297.763,Z 396.888,A -85,B 0,C 180,E1 -16521.772,E2 -16521.772} C_VEL
LIN {X 0,Y 294.914,Z 397.249,A -85,B 0,C 180,E1 -16523.607,E2 -16523.607} C_VEL
LIN {X 0,Y 292.481,Z 397.552,A -85,B 0,C 180,E1 -16525.096,E2 -16525.096} C_VEL
LIN {X 0,Y 291.426,Z 397.682,A -85,B 0,C 180,E1 -16526.249,E2 -16526.249} C_VEL
LIN {X 0,Y 291.334,Z 397.692,A -85,B 0,C 180,E1 -16526.64,E2 -16526.64} C_VEL
LIN {X 0,Y 291.391,Z 397.686,A -85,B 0,C 180,E1 -16530.26,E2 -16530.26} C_VEL
LIN {X 0,Y 291.421,Z 397.682,A -85,B 0,C 180,E1 -16534.272,E2 -16534.272} C_VEL
LIN {X 0,Y 291.394,Z 397.685,A -85,B 0,C 180,E1 -16537.3,E2 -16537.3} C_VEL
LIN {X 0,Y 291.468,Z 397.675,A -85,B 0,C 180,E1 -16540.271,E2 -16540.271} C_VEL
LIN {X 0,Y 291.559,Z 397.664,A -85,B 0,C 180,E1 -16544.624,E2 -16544.624} C_VEL
LIN {X 0,Y 291.541,Z 397.667,A -85,B 0,C 180,E1 -16548.881,E2 -16548.881} C_VEL
LIN {X 0,Y 291.714,Z 397.647,A -85,B 0,C 180,E1 -16551.689,E2 -16551.689} C_VEL
LIN {X 0,Y 291.636,Z 397.656,A -85,B 0,C 180,E1 -16554.468,E2 -16554.468} C_VEL
LIN {X 0,Y 291.893,Z 397.618,A -85,B 0,C 180,E1 -16558.62,E2 -16558.62} C_VEL
LIN {X 0,Y 291.893,Z 397.623,A -85,B 0,C 180,E1 -16561.38,E2 -16561.38} C_VEL
LIN {X 0,Y 291.729,Z 397.641,A -85,B 0,C 180,E1 -16566.918,E2 -16566.918} C_VEL
LIN {X 0,Y 291.577,Z 397.665,A -85,B 0,C 180,E1 -16569.714,E2 -16569.714} C_VEL
LIN {X 0,Y 291.527,Z 397.671,A -85,B 0,C 180,E1 -16573.95,E2 -16573.95} C_VEL
LIN {X 0,Y 291.491,Z 397.67,A -85,B 0,C 180,E1 -16576.818,E2 -16576.818} C_VEL
LIN {X 0,Y 291.454,Z 397.68,A -85,B 0,C 180,E1 -16579.875,E2 -16579.875} C_VEL
LIN {X 0,Y 291.404,Z 397.685,A -85,B 0,C 180,E1 -16584.205,E2 -16584.205} C_VEL
LIN {X 0,Y 291.423,Z 397.686,A -85,B 0,C 180,E1 -16587.271,E2 -16587.271} C_VEL
LIN {X 0,Y 291.338,Z 397.691,A -85,B 0,C 180,E1 -16590.437,E2 -16590.437} C_VEL
LIN {X 0,Y 291.348,Z 397.692,A -85,B 0,C 180,E1 -16593.698,E2 -16593.698} C_VEL
LIN {X 0,Y 291.376,Z 397.691,A -85,B 0,C 180,E1 -16597.253,E2 -16597.253} C_VEL
LIN {X 0,Y 291.336,Z 397.693,A -85,B 0,C 180,E1 -16600.642,E2 -16600.642} C_VEL
LIN {X 0,Y 291.316,Z 397.696,A -85,B 0,C 180,E1 -16604.397,E2 -16604.397} C_VEL
LIN {X 0,Y 291.33,Z 397.696,A -85,B 0,C 180,E1 -16608.404,E2 -16608.404} C_VEL
LIN {X 0,Y 291.356,Z 397.694,A -85,B 0,C 180,E1 -16611.158,E2 -16611.158} C_VEL
LIN {X 0,Y 291.364,Z 397.691,A -85,B 0,C 180,E1 -16614.626,E2 -16614.626} C_VEL
LIN {X 0,Y 291.407,Z 397.83,A -85,B 0,C 180,E1 -16615.654,E2 -16615.654} C_VEL
LIN {X 0,Y 293.836,Z 408.359,A -85,B 0,C 180,E1 -16619.435,E2 -16619.435} C_VEL
LIN {X 0,Y 295.6,Z 417.085,A -85,B 0,C 180,E1 -16622.371,E2 -16622.371} C_VEL
LIN {X 0,Y 299.436,Z 427.211,A -85,B 0,C 180,E1 -16623.019,E2 -16623.019} C_VEL
LIN {X 0,Y 304.085,Z 454.057,A -85,B 0,C 180,E1 -16624.152,E2 -16624.152} C_VEL
LIN {X 0,Y 304.842,Z 460.604,A -85,B 0,C 180,E1 -16624.388,E2 -16624.388} C_VEL
LIN {X 0,Y 303.08,Z 525.307,A -85,B 0,C 180,E1 -16625.922,E2 -16625.922} C_VEL
LIN {X 0,Y 302.128,Z 539.241,A -85,B 0,C 180,E1 -16626.524,E2 -16626.524} C_VEL
LIN {X 0,Y 300.885,Z 551.699,A -85,B 0,C 180,E1 -16627.331,E2 -16627.331} C_VEL
LIN {X 0,Y 299.491,Z 562.808,A -85,B 0,C 180,E1 -16628.309,E2 -16628.309} C_VEL
LIN {X 0,Y 297.823,Z 574.38,A -85,B 0,C 180,E1 -16629.63,E2 -16629.63} C_VEL
LIN {X 0,Y 296.053,Z 584.799,A -85,B 0,C 180,E1 -16631.128,E2 -16631.128} C_VEL
LIN {X 0,Y 294.581,Z 594.049,A -85,B 0,C 180,E1 -16632.799,E2 -16632.799} C_VEL
LIN {X 0,Y 293.128,Z 602.563,A -85,B 0,C 180,E1 -16634.708,E2 -16634.708} C_VEL
LIN {X 0,Y 291.703,Z 609.986,A -85,B 0,C 180,E1 -16636.768,E2 -16636.768} C_VEL
LIN {X 0,Y 290.743,Z 615.952,A -85,B 0,C 180,E1 -16638.85,E2 -16638.85} C_VEL
LIN {X 0,Y 290.054,Z 620.667,A -85,B 0,C 180,E1 -16640.938,E2 -16640.938} C_VEL
LIN {X 0,Y 289.608,Z 624.271,A -85,B 0,C 180,E1 -16643.03,E2 -16643.03} C_VEL
LIN {X 0,Y 289.428,Z 626.328,A -85,B 0,C 180,E1 -16644.612,E2 -16644.612} C_VEL
LIN {X 0,Y 289.427,Z 628.521,A -85,B 0,C 180,E1 -16647.216,E2 -16647.216} C_VEL
LIN {X 0,Y 289.399,Z 629.128,A -85,B 0,C 180,E1 -16648.608,E2 -16648.608} C_VEL
LIN {X 0,Y 289.401,Z 629.341,A -85,B 0,C 180,E1 -16650,E2 -16650} C_VEL
LIN {X 0,Y 289.398,Z 629.12,A -85,B 0,C 180,E1 -16651.391,E2 -16651.391} C_VEL
LIN {X 0,Y 289.427,Z 628.51,A -85,B 0,C 180,E1 -16652.783,E2 -16652.783} C_VEL
LIN {X 0,Y 289.477,Z 626.107,A -85,B 0,C 180,E1 -16655.573,E2 -16655.573} C_VEL
LIN {X 0,Y 289.729,Z 623.164,A -85,B 0,C 180,E1 -16657.667,E2 -16657.667} C_VEL
LIN {X 0,Y 290.255,Z 619.185,A -85,B 0,C 180,E1 -16659.758,E2 -16659.758} C_VEL
LIN {X 0,Y 291.132,Z 613.067,A -85,B 0,C 180,E1 -16662.194,E2 -16662.194} C_VEL
LIN {X 0,Y 292.375,Z 606.39,A -85,B 0,C 180,E1 -16664.264,E2 -16664.264} C_VEL
LIN {X 0,Y 293.843,Z 598.105,A -85,B 0,C 180,E1 -16666.322,E2 -16666.322} C_VEL
LIN {X 0,Y 295.265,Z 589.609,A -85,B 0,C 180,E1 -16668.025,E2 -16668.025} C_VEL
LIN {X 0,Y 296.955,Z 579.113,A -85,B 0,C 180,E1 -16669.709,E2 -16669.709} C_VEL
LIN {X 0,Y 298.814,Z 567.302,A -85,B 0,C 180,E1 -16671.199,E2 -16671.199} C_VEL
LIN {X 0,Y 300.385,Z 555.406,A -85,B 0,C 180,E1 -16672.346,E2 -16672.346} C_VEL
LIN {X 0,Y 301.684,Z 543.024,A -85,B 0,C 180,E1 -16673.239,E2 -16673.239} C_VEL
LIN {X 0,Y 302.789,Z 530.28,A -85,B 0,C 180,E1 -16673.875,E2 -16673.875} C_VEL
LIN {X 0,Y 303.381,Z 516.819,A -85,B 0,C 180,E1 -16674.279,E2 -16674.279} C_VEL
LIN {X 0,Y 304.686,Z 458.719,A -85,B 0,C 180,E1 -16675.647,E2 -16675.647} C_VEL
LIN {X 0,Y 300.641,Z 433.914,A -85,B 0,C 180,E1 -16676.661,E2 -16676.661} C_VEL
LIN {X 0,Y 298.882,Z 425.399,A -85,B 0,C 180,E1 -16677.053,E2 -16677.053} C_VEL
LIN {X 0,Y 295.536,Z 416.821,A -85,B 0,C 180,E1 -16677.653,E2 -16677.653} C_VEL
LIN {X 0,Y 293.801,Z 408.306,A -85,B 0,C 180,E1 -16680.553,E2 -16680.553} C_VEL
LIN {X 0,Y 291.537,Z 398.471,A -85,B 0,C 180,E1 -16684.076,E2 -16684.076} C_VEL
LIN {X 0,Y 291.389,Z 397.688,A -85,B 0,C 180,E1 -16684.399,E2 -16684.399} C_VEL
LIN {X 0,Y 291.377,Z 397.69,A -85,B 0,C 180,E1 -16687.254,E2 -16687.254} C_VEL
LIN {X 0,Y 291.334,Z 397.696,A -85,B 0,C 180,E1 -16690.642,E2 -16690.642} C_VEL
LIN {X 0,Y 291.314,Z 397.695,A -85,B 0,C 180,E1 -16694.397,E2 -16694.397} C_VEL
LIN {X 0,Y 291.328,Z 397.695,A -85,B 0,C 180,E1 -16698.404,E2 -16698.404} C_VEL
LIN {X 0,Y 291.349,Z 397.691,A -85,B 0,C 180,E1 -16701.158,E2 -16701.158} C_VEL
LIN {X 0,Y 291.362,Z 397.692,A -85,B 0,C 180,E1 -16704.626,E2 -16704.626} C_VEL
LIN {X 0,Y 291.371,Z 397.688,A -85,B 0,C 180,E1 -16707.951,E2 -16707.951} C_VEL
LIN {X 0,Y 291.379,Z 397.688,A -85,B 0,C 180,E1 -16711.158,E2 -16711.158} C_VEL
LIN {X 0,Y 291.416,Z 397.685,A -85,B 0,C 180,E1 -16714.272,E2 -16714.272} C_VEL
LIN {X 0,Y 291.391,Z 397.686,A -85,B 0,C 180,E1 -16717.3,E2 -16717.3} C_VEL
LIN {X 0,Y 291.46,Z 397.679,A -85,B 0,C 180,E1 -16720.27,E2 -16720.27} C_VEL
LIN {X 0,Y 291.556,Z 397.665,A -85,B 0,C 180,E1 -16724.624,E2 -16724.624} C_VEL
LIN {X 0,Y 291.539,Z 397.667,A -85,B 0,C 180,E1 -16728.881,E2 -16728.881} C_VEL
LIN {X 0,Y 291.67,Z 397.65,A -85,B 0,C 180,E1 -16731.687,E2 -16731.687} C_VEL
LIN {X 0,Y 291.626,Z 397.656,A -85,B 0,C 180,E1 -16734.468,E2 -16734.468} C_VEL
LIN {X 0,Y 291.89,Z 397.625,A -85,B 0,C 180,E1 -16738.62,E2 -16738.62} C_VEL
LIN {X 0,Y 291.892,Z 397.619,A -85,B 0,C 180,E1 -16741.38,E2 -16741.38} C_VEL
LIN {X 0,Y 291.749,Z 397.638,A -85,B 0,C 180,E1 -16746.918,E2 -16746.918} C_VEL
LIN {X 0,Y 291.631,Z 397.658,A -85,B 0,C 180,E1 -16749.712,E2 -16749.712} C_VEL
LIN {X 0,Y 291.524,Z 397.673,A -85,B 0,C 180,E1 -16753.95,E2 -16753.95} C_VEL
LIN {X 0,Y 291.489,Z 397.669,A -85,B 0,C 180,E1 -16756.818,E2 -16756.818} C_VEL
LIN {X 0,Y 291.454,Z 397.682,A -85,B 0,C 180,E1 -16759.876,E2 -16759.876} C_VEL
LIN {X 0,Y 291.402,Z 397.686,A -85,B 0,C 180,E1 -16764.205,E2 -16764.205} C_VEL
LIN {X 0,Y 291.424,Z 397.681,A -85,B 0,C 180,E1 -16767.272,E2 -16767.272} C_VEL
LIN {X 0,Y 291.339,Z 397.691,A -85,B 0,C 180,E1 -16770.437,E2 -16770.437} C_VEL
LIN {X 0,Y 291.347,Z 397.693,A -85,B 0,C 180,E1 -16773.698,E2 -16773.698} C_VEL
LIN {X 0,Y 291.398,Z 397.686,A -85,B 0,C 180,E1 -16777.26,E2 -16777.26} C_VEL
LIN {X 0,Y 291.374,Z 397.686,A -85,B 0,C 180,E1 -16780.636,E2 -16780.636} C_VEL
LIN {X 0,Y 291.291,Z 397.697,A -85,B 0,C 180,E1 -16784.402,E2 -16784.402} C_VEL
LIN {X 0,Y 291.328,Z 397.695,A -85,B 0,C 180,E1 -16788.404,E2 -16788.404} C_VEL
LIN {X 0,Y 291.355,Z 397.694,A -85,B 0,C 180,E1 -16791.159,E2 -16791.159} C_VEL
LIN {X 0,Y 291.363,Z 397.691,A -85,B 0,C 180,E1 -16794.626,E2 -16794.626} C_VEL
LIN {X 0,Y 291.376,Z 397.686,A -85,B 0,C 180,E1 -16799.267,E2 -16799.267} C_VEL
LIN {X 0,Y 293.177,Z 405.318,A -85,B 0,C 180,E1 -16802.212,E2 -16802.212} C_VEL
LIN {X 0,Y 301.247,Z 424.514,A -85,B 0,C 180,E1 -16803.527,E2 -16803.527} C_VEL
LIN {X 0,Y 303.746,Z 431.389,A -85,B 0,C 180,E1 -16803.942,E2 -16803.942} C_VEL
LIN {X 0,Y 305.317,Z 439.849,A -85,B 0,C 180,E1 -16804.304,E2 -16804.304} C_VEL
LIN {X 0,Y 303.436,Z 511.603,A -85,B 0,C 180,E1 -16805.998,E2 -16805.998} C_VEL
LIN {X 0,Y 302.567,Z 524.979,A -85,B 0,C 180,E1 -16806.561,E2 -16806.561} C_VEL
LIN {X 0,Y 301.446,Z 537.737,A -85,B 0,C 180,E1 -16807.376,E2 -16807.376} C_VEL
LIN {X 0,Y 300.132,Z 549.066,A -85,B 0,C 180,E1 -16808.358,E2 -16808.358} C_VEL
LIN {X 0,Y 298.552,Z 560.712,A -85,B 0,C 180,E1 -16809.683,E2 -16809.683} C_VEL
LIN {X 0,Y 296.968,Z 571.221,A -85,B 0,C 180,E1 -16811.198,E2 -16811.198} C_VEL
LIN {X 0,Y 295.651,Z 579.707,A -85,B 0,C 180,E1 -16812.714,E2 -16812.714} C_VEL
LIN {X 0,Y 294.178,Z 587.578,A -85,B 0,C 180,E1 -16814.409,E2 -16814.409} C_VEL
LIN {X 0,Y 292.705,Z 595.269,A -85,B 0,C 180,E1 -16816.461,E2 -16816.461} C_VEL
LIN {X 0,Y 291.416,Z 602.328,A -85,B 0,C 180,E1 -16818.876,E2 -16818.876} C_VEL
LIN {X 0,Y 290.571,Z 607.028,A -85,B 0,C 180,E1 -16820.955,E2 -16820.955} C_VEL
LIN {X 0,Y 290.029,Z 610.624,A -85,B 0,C 180,E1 -16823.041,E2 -16823.041} C_VEL
LIN {X 0,Y 289.805,Z 612.481,A -85,B 0,C 180,E1 -16824.434,E2 -16824.434} C_VEL
LIN {X 0,Y 289.66,Z 613.877,A -85,B 0,C 180,E1 -16825.826,E2 -16825.826} C_VEL
LIN {X 0,Y 289.54,Z 614.87,A -85,B 0,C 180,E1 -16827.218,E2 -16827.218} C_VEL
LIN {X 0,Y 289.407,Z 615.713,A -85,B 0,C 180,E1 -16830,E2 -16830} C_VEL
LIN {X 0,Y 289.44,Z 615.52,A -85,B 0,C 180,E1 -16831.392,E2 -16831.392} C_VEL
LIN {X 0,Y 289.54,Z 614.933,A -85,B 0,C 180,E1 -16832.783,E2 -16832.783} C_VEL
LIN {X 0,Y 289.657,Z 613.965,A -85,B 0,C 180,E1 -16834.175,E2 -16834.175} C_VEL
LIN {X 0,Y 289.906,Z 611.678,A -85,B 0,C 180,E1 -16836.31,E2 -16836.31} C_VEL
LIN {X 0,Y 290.378,Z 608.541,A -85,B 0,C 180,E1 -16838.35,E2 -16838.35} C_VEL
LIN {X 0,Y 291.076,Z 604.284,A -85,B 0,C 180,E1 -16840.433,E2 -16840.433} C_VEL
LIN {X 0,Y 292.25,Z 597.838,A -85,B 0,C 180,E1 -16842.853,E2 -16842.853} C_VEL
LIN {X 0,Y 293.536,Z 590.754,A -85,B 0,C 180,E1 -16844.915,E2 -16844.915} C_VEL
LIN {X 0,Y 295.268,Z 581.923,A -85,B 0,C 180,E1 -16846.953,E2 -16846.953} C_VEL
LIN {X 0,Y 296.81,Z 572.486,A -85,B 0,C 180,E1 -16848.712,E2 -16848.712} C_VEL
LIN {X 0,Y 298.231,Z 562.83,A -85,B 0,C 180,E1 -16850.161,E2 -16850.161} C_VEL
LIN {X 0,Y 299.879,Z 551.662,A -85,B 0,C 180,E1 -16851.481,E2 -16851.481} C_VEL
LIN {X 0,Y 301.344,Z 539.126,A -85,B 0,C 180,E1 -16852.633,E2 -16852.633} C_VEL
LIN {X 0,Y 302.514,Z 526.18,A -85,B 0,C 180,E1 -16853.489,E2 -16853.489} C_VEL
LIN {X 0,Y 303.343,Z 513.401,A -85,B 0,C 180,E1 -16854.056,E2 -16854.056} C_VEL
LIN {X 0,Y 304.256,Z 483.254,A -85,B 0,C 180,E1 -16854.799,E2 -16854.799} C_VEL
LIN {X 0,Y 305.261,Z 439.255,A -85,B 0,C 180,E1 -16855.834,E2 -16855.834} C_VEL
LIN {X 0,Y 303.385,Z 430.192,A -85,B 0,C 180,E1 -16856.241,E2 -16856.241} C_VEL
LIN {X 0,Y 296.345,Z 412.643,A -85,B 0,C 180,E1 -16857.387,E2 -16857.387} C_VEL
LIN {X 0,Y 293.123,Z 405.094,A -85,B 0,C 180,E1 -16857.933,E2 -16857.933} C_VEL
LIN {X 0,Y 291.381,Z 397.692,A -85,B 0,C 180,E1 -16860.834,E2 -16860.834} C_VEL
LIN {X 0,Y 291.364,Z 397.689,A -85,B 0,C 180,E1 -16865.374,E2 -16865.374} C_VEL
LIN {X 0,Y 291.356,Z 397.693,A -85,B 0,C 180,E1 -16868.842,E2 -16868.842} C_VEL
LIN {X 0,Y 291.323,Z 397.698,A -85,B 0,C 180,E1 -16872.492,E2 -16872.492} C_VEL
LIN {X 0,Y 291.342,Z 397.694,A -85,B 0,C 180,E1 -16876.36,E2 -16876.36} C_VEL
LIN {X 0,Y 291.388,Z 397.678,A -85,B 0,C 180,E1 -16880.632,E2 -16880.632} C_VEL
LIN {X 0,Y 291.43,Z 397.682,A -85,B 0,C 180,E1 -16882.923,E2 -16882.923} C_VEL
LIN {X 0,Y 291.334,Z 397.692,A -85,B 0,C 180,E1 -16886.64,E2 -16886.64} C_VEL
LIN {X 0,Y 290.642,Z 397.781,A -85,B 0,C 180,E1 -16887.795,E2 -16887.795} C_VEL
LIN {X 0,Y 287.766,Z 398.137,A -85,B 0,C 180,E1 -16889.676,E2 -16889.676} C_VEL
LIN {X 0,Y 285.388,Z 398.432,A -85,B 0,C 180,E1 -16891.203,E2 -16891.203} C_VEL
LIN {X 0,Y 284.437,Z 398.556,A -85,B 0,C 180,E1 -16892.386,E2 -16892.386} C_VEL
LIN {X 0,Y 284.397,Z 398.558,A -85,B 0,C 180,E1 -16892.786,E2 -16892.786} C_VEL
LIN {X 0,Y 284.374,Z 398.561,A -85,B 0,C 180,E1 -16896.707,E2 -16896.707} C_VEL
LIN {X 0,Y 284.41,Z 398.551,A -85,B 0,C 180,E1 -16901.262,E2 -16901.262} C_VEL
LIN {X 0,Y 284.496,Z 398.545,A -85,B 0,C 180,E1 -16904.459,E2 -16904.459} C_VEL
LIN {X 0,Y 284.493,Z 398.546,A -85,B 0,C 180,E1 -16908.602,E2 -16908.602} C_VEL
LIN {X 0,Y 284.664,Z 398.524,A -85,B 0,C 180,E1 -16911.481,E2 -16911.481} C_VEL
LIN {X 0,Y 284.607,Z 398.532,A -85,B 0,C 180,E1 -16914.331,E2 -16914.331} C_VEL
LIN {X 0,Y 284.859,Z 398.494,A -85,B 0,C 180,E1 -16918.586,E2 -16918.586} C_VEL
LIN {X 0,Y 284.859,Z 398.5,A -85,B 0,C 180,E1 -16921.414,E2 -16921.414} C_VEL
LIN {X 0,Y 284.68,Z 398.52,A -85,B 0,C 180,E1 -16927.09,E2 -16927.09} C_VEL
LIN {X 0,Y 284.522,Z 398.541,A -85,B 0,C 180,E1 -16929.957,E2 -16929.957} C_VEL
LIN {X 0,Y 284.487,Z 398.546,A -85,B 0,C 180,E1 -16934.302,E2 -16934.302} C_VEL
LIN {X 0,Y 284.43,Z 398.551,A -85,B 0,C 180,E1 -16937.248,E2 -16937.248} C_VEL
LIN {X 0,Y 284.383,Z 398.559,A -85,B 0,C 180,E1 -16940.242,E2 -16940.242} C_VEL
LIN {X 0,Y 284.373,Z 398.562,A -85,B 0,C 180,E1 -16943.875,E2 -16943.875} C_VEL
LIN {X 0,Y 284.399,Z 398.56,A -85,B 0,C 180,E1 -16947.173,E2 -16947.173} C_VEL
LIN {X 0,Y 284.297,Z 398.573,A -85,B 0,C 180,E1 -16951.274,E2 -16951.274} C_VEL
LIN {X 0,Y 284.344,Z 398.567,A -85,B 0,C 180,E1 -16955.348,E2 -16955.348} C_VEL
LIN {X 0,Y 284.311,Z 398.567,A -85,B 0,C 180,E1 -16958.169,E2 -16958.169} C_VEL
LIN {X 0,Y 284.272,Z 398.573,A -85,B 0,C 180,E1 -16962.124,E2 -16962.124} C_VEL
LIN {X 0,Y 284.271,Z 398.574,A -85,B 0,C 180,E1 -16966.192,E2 -16966.192} C_VEL
LIN {X 0,Y 284.309,Z 398.569,A -85,B 0,C 180,E1 -16970.024,E2 -16970.024} C_VEL
LIN {X 0,Y 284.335,Z 398.568,A -85,B 0,C 180,E1 -16973.614,E2 -16973.614} C_VEL
LIN {X 0,Y 284.328,Z 398.591,A -85,B 0,C 180,E1 -16975.002,E2 -16975.002} C_VEL
LIN {X 0,Y 286.57,Z 408.228,A -85,B 0,C 180,E1 -16978.59,E2 -16978.59} C_VEL
LIN {X 0,Y 288.412,Z 417.048,A -85,B 0,C 180,E1 -16981.624,E2 -16981.624} C_VEL
LIN {X 0,Y 293.264,Z 429.215,A -85,B 0,C 180,E1 -16982.461,E2 -16982.461} C_VEL
LIN {X 0,Y 297.786,Z 455.561,A -85,B 0,C 180,E1 -16983.607,E2 -16983.607} C_VEL
LIN {X 0,Y 298.443,Z 461.805,A -85,B 0,C 180,E1 -16983.833,E2 -16983.833} C_VEL
LIN {X 0,Y 296.62,Z 525.153,A -85,B 0,C 180,E1 -16985.363,E2 -16985.363} C_VEL
LIN {X 0,Y 295.636,Z 539.083,A -85,B 0,C 180,E1 -16985.977,E2 -16985.977} C_VEL
LIN {X 0,Y 294.367,Z 551.539,A -85,B 0,C 180,E1 -16986.8,E2 -16986.8} C_VEL
LIN {X 0,Y 292.909,Z 562.645,A -85,B 0,C 180,E1 -16987.796,E2 -16987.796} C_VEL
LIN {X 0,Y 291.178,Z 574.216,A -85,B 0,C 180,E1 -16989.144,E2 -16989.144} C_VEL
LIN {X 0,Y 289.326,Z 584.634,A -85,B 0,C 180,E1 -16990.672,E2 -16990.672} C_VEL
LIN {X 0,Y 287.876,Z 592.997,A -85,B 0,C 180,E1 -16992.199,E2 -16992.199} C_VEL
LIN {X 0,Y 286.518,Z 601.022,A -85,B 0,C 180,E1 -16993.981,E2 -16993.981} C_VEL
LIN {X 0,Y 285.028,Z 608.701,A -85,B 0,C 180,E1 -16996.089,E2 -16996.089} C_VEL
LIN {X 0,Y 284.028,Z 613.965,A -85,B 0,C 180,E1 -16997.858,E2 -16997.858} C_VEL
LIN {X 0,Y 283.221,Z 619.068,A -85,B 0,C 180,E1 -16999.997,E2 -16999.997} C_VEL
LIN {X 0,Y 282.686,Z 623.033,A -85,B 0,C 180,E1 -17002.141,E2 -17002.141} C_VEL
LIN {X 0,Y 282.331,Z 626.384,A -85,B 0,C 180,E1 -17004.694,E2 -17004.694} C_VEL
LIN {X 0,Y 282.333,Z 628.354,A -85,B 0,C 180,E1 -17007.146,E2 -17007.146} C_VEL
LIN {X 0,Y 282.322,Z 628.961,A -85,B 0,C 180,E1 -17008.573,E2 -17008.573} C_VEL
LIN {X 0,Y 282.322,Z 629.174,A -85,B 0,C 180,E1 -17010,E2 -17010} C_VEL
LIN {X 0,Y 282.322,Z 628.954,A -85,B 0,C 180,E1 -17011.426,E2 -17011.426} C_VEL
LIN {X 0,Y 282.333,Z 628.342,A -85,B 0,C 180,E1 -17012.853,E2 -17012.853} C_VEL
LIN {X 0,Y 282.386,Z 625.939,A -85,B 0,C 180,E1 -17015.713,E2 -17015.713} C_VEL
LIN {X 0,Y 282.686,Z 622.996,A -85,B 0,C 180,E1 -17017.859,E2 -17017.859} C_VEL
LIN {X 0,Y 283.22,Z 619.016,A -85,B 0,C 180,E1 -17020.003,E2 -17020.003} C_VEL
LIN {X 0,Y 284.164,Z 612.897,A -85,B 0,C 180,E1 -17022.498,E2 -17022.498} C_VEL
LIN {X 0,Y 285.476,Z 606.22,A -85,B 0,C 180,E1 -17024.616,E2 -17024.616} C_VEL
LIN {X 0,Y 287.023,Z 597.936,A -85,B 0,C 180,E1 -17026.721,E2 -17026.721} C_VEL
LIN {X 0,Y 288.495,Z 589.439,A -85,B 0,C 180,E1 -17028.463,E2 -17028.463} C_VEL
LIN {X 0,Y 290.267,Z 578.942,A -85,B 0,C 180,E1 -17030.183,E2 -17030.183} C_VEL
LIN {X 0,Y 292.177,Z 567.129,A -85,B 0,C 180,E1 -17031.705,E2 -17031.705} C_VEL
LIN {X 0,Y 293.845,Z 555.233,A -85,B 0,C 180,E1 -17032.871,E2 -17032.871} C_VEL
LIN {X 0,Y 295.177,Z 542.849,A -85,B 0,C 180,E1 -17033.783,E2 -17033.783} C_VEL
LIN {X 0,Y 296.32,Z 530.102,A -85,B 0,C 180,E1 -17034.429,E2 -17034.429} C_VEL
LIN {X 0,Y 296.944,Z 516.631,A -85,B 0,C 180,E1 -17034.841,E2 -17034.841} C_VEL
LIN {X 0,Y 298.301,Z 459.741,A -85,B 0,C 180,E1 -17036.205,E2 -17036.205} C_VEL
LIN {X 0,Y 294.388,Z 435.601,A -85,B 0,C 180,E1 -17037.223,E2 -17037.223} C_VEL
LIN {X 0,Y 292.878,Z 428.189,A -85,B 0,C 180,E1 -17037.574,E2 -17037.574} C_VEL
LIN {X 0,Y 288.345,Z 416.695,A -85,B 0,C 180,E1 -17038.385,E2 -17038.385} C_VEL
LIN {X 0,Y 286.293,Z 406.896,A -85,B 0,C 180,E1 -17041.856,E2 -17041.856} C_VEL
LIN {X 0,Y 284.326,Z 398.569,A -85,B 0,C 180,E1 -17044.998,E2 -17044.998} C_VEL
LIN {X 0,Y 284.313,Z 398.569,A -85,B 0,C 180,E1 -17048.169,E2 -17048.169} C_VEL
LIN {X 0,Y 284.27,Z 398.573,A -85,B 0,C 180,E1 -17052.124,E2 -17052.124} C_VEL
LIN {X 0,Y 284.269,Z 398.573,A -85,B 0,C 180,E1 -17056.192,E2 -17056.192} C_VEL
LIN {X 0,Y 284.307,Z 398.567,A -85,B 0,C 180,E1 -17060.024,E2 -17060.024} C_VEL
LIN {X 0,Y 284.331,Z 398.565,A -85,B 0,C 180,E1 -17063.614,E2 -17063.614} C_VEL
LIN {X 0,Y 284.308,Z 398.569,A -85,B 0,C 180,E1 -17067.19,E2 -17067.19} C_VEL
LIN {X 0,Y 284.356,Z 398.564,A -85,B 0,C 180,E1 -17070.376,E2 -17070.376} C_VEL
LIN {X 0,Y 284.377,Z 398.559,A -85,B 0,C 180,E1 -17073.586,E2 -17073.586} C_VEL
LIN {X 0,Y 284.37,Z 398.562,A -85,B 0,C 180,E1 -17076.707,E2 -17076.707} C_VEL
LIN {X 0,Y 284.405,Z 398.555,A -85,B 0,C 180,E1 -17081.262,E2 -17081.262} C_VEL
LIN {X 0,Y 284.494,Z 398.545,A -85,B 0,C 180,E1 -17084.459,E2 -17084.459} C_VEL
LIN {X 0,Y 284.491,Z 398.547,A -85,B 0,C 180,E1 -17088.602,E2 -17088.602} C_VEL
LIN {X 0,Y 284.624,Z 398.527,A -85,B 0,C 180,E1 -17091.48,E2 -17091.48} C_VEL
LIN {X 0,Y 284.596,Z 398.533,A -85,B 0,C 180,E1 -17094.331,E2 -17094.331} C_VEL
LIN {X 0,Y 284.857,Z 398.502,A -85,B 0,C 180,E1 -17098.586,E2 -17098.586} C_VEL
LIN {X 0,Y 284.858,Z 398.495,A -85,B 0,C 180,E1 -17101.414,E2 -17101.414} C_VEL
LIN {X 0,Y 284.701,Z 398.516,A -85,B 0,C 180,E1 -17107.09,E2 -17107.09} C_VEL
LIN {X 0,Y 284.568,Z 398.54,A -85,B 0,C 180,E1 -17109.955,E2 -17109.955} C_VEL
LIN {X 0,Y 284.483,Z 398.549,A -85,B 0,C 180,E1 -17114.303,E2 -17114.303} C_VEL
LIN {X 0,Y 284.428,Z 398.549,A -85,B 0,C 180,E1 -17117.248,E2 -17117.248} C_VEL
LIN {X 0,Y 284.383,Z 398.56,A -85,B 0,C 180,E1 -17120.242,E2 -17120.242} C_VEL
LIN {X 0,Y 284.371,Z 398.565,A -85,B 0,C 180,E1 -17123.876,E2 -17123.876} C_VEL
LIN {X 0,Y 284.399,Z 398.556,A -85,B 0,C 180,E1 -17127.174,E2 -17127.174} C_VEL
LIN {X 0,Y 284.298,Z 398.569,A -85,B 0,C 180,E1 -17131.274,E2 -17131.274} C_VEL
LIN {X 0,Y 284.363,Z 398.562,A -85,B 0,C 180,E1 -17135.354,E2 -17135.354} C_VEL
LIN {X 0,Y 284.329,Z 398.566,A -85,B 0,C 180,E1 -17138.167,E2 -17138.167} C_VEL
LIN {X 0,Y 284.291,Z 398.573,A -85,B 0,C 180,E1 -17141.872,E2 -17141.872} C_VEL
LIN {X 0,Y 284.256,Z 398.574,A -85,B 0,C 180,E1 -17146.189,E2 -17146.189} C_VEL
LIN {X 0,Y 284.308,Z 398.57,A -85,B 0,C 180,E1 -17150.024,E2 -17150.024} C_VEL
LIN {X 0,Y 284.334,Z 398.567,A -85,B 0,C 180,E1 -17153.614,E2 -17153.614} C_VEL
LIN {X 0,Y 284.31,Z 398.571,A -85,B 0,C 180,E1 -17157.19,E2 -17157.19} C_VEL
LIN {X 0,Y 284.375,Z 398.729,A -85,B 0,C 180,E1 -17158.809,E2 -17158.809} C_VEL
LIN {X 0,Y 285.912,Z 405.373,A -85,B 0,C 180,E1 -17161.438,E2 -17161.438} C_VEL
LIN {X 0,Y 294.575,Z 425.503,A -85,B 0,C 180,E1 -17162.901,E2 -17162.901} C_VEL
LIN {X 0,Y 297.75,Z 434.567,A -85,B 0,C 180,E1 -17163.455,E2 -17163.455} C_VEL
LIN {X 0,Y 298.896,Z 440.571,A -85,B 0,C 180,E1 -17163.724,E2 -17163.724} C_VEL
LIN {X 0,Y 296.986,Z 511.786,A -85,B 0,C 180,E1 -17165.443,E2 -17165.443} C_VEL
LIN {X 0,Y 296.09,Z 525.155,A -85,B 0,C 180,E1 -17166.016,E2 -17166.016} C_VEL
LIN {X 0,Y 294.916,Z 537.912,A -85,B 0,C 180,E1 -17166.846,E2 -17166.846} C_VEL
LIN {X 0,Y 293.569,Z 549.238,A -85,B 0,C 180,E1 -17167.849,E2 -17167.849} C_VEL
LIN {X 0,Y 291.903,Z 560.883,A -85,B 0,C 180,E1 -17169.199,E2 -17169.199} C_VEL
LIN {X 0,Y 290.164,Z 571.979,A -85,B 0,C 180,E1 -17170.842,E2 -17170.842} C_VEL
LIN {X 0,Y 288.56,Z 581.569,A -85,B 0,C 180,E1 -17172.641,E2 -17172.641} C_VEL
LIN {X 0,Y 286.729,Z 590.486,A -85,B 0,C 180,E1 -17174.723,E2 -17174.723} C_VEL
LIN {X 0,Y 285.388,Z 597.659,A -85,B 0,C 180,E1 -17176.833,E2 -17176.833} C_VEL
LIN {X 0,Y 284.428,Z 602.497,A -85,B 0,C 180,E1 -17178.599,E2 -17178.599} C_VEL
LIN {X 0,Y 283.542,Z 607.197,A -85,B 0,C 180,E1 -17180.729,E2 -17180.729} C_VEL
LIN {X 0,Y 282.982,Z 610.792,A -85,B 0,C 180,E1 -17182.867,E2 -17182.867} C_VEL
LIN {X 0,Y 282.727,Z 612.649,A -85,B 0,C 180,E1 -17184.294,E2 -17184.294} C_VEL
LIN {X 0,Y 282.584,Z 614.044,A -85,B 0,C 180,E1 -17185.721,E2 -17185.721} C_VEL
LIN {X 0,Y 282.472,Z 615.037,A -85,B 0,C 180,E1 -17187.148,E2 -17187.148} C_VEL
LIN {X 0,Y 282.328,Z 615.88,A -85,B 0,C 180,E1 -17190,E2 -17190} C_VEL
LIN {X 0,Y 282.364,Z 615.687,A -85,B 0,C 180,E1 -17191.427,E2 -17191.427} C_VEL
LIN {X 0,Y 282.472,Z 615.099,A -85,B 0,C 180,E1 -17192.853,E2 -17192.853} C_VEL
LIN {X 0,Y 282.582,Z 614.131,A -85,B 0,C 180,E1 -17194.279,E2 -17194.279} C_VEL
LIN {X 0,Y 282.817,Z 612.082,A -85,B 0,C 180,E1 -17196.277,E2 -17196.277} C_VEL
LIN {X 0,Y 283.356,Z 608.707,A -85,B 0,C 180,E1 -17198.559,E2 -17198.559} C_VEL
LIN {X 0,Y 284.075,Z 604.45,A -85,B 0,C 180,E1 -17200.694,E2 -17200.694} C_VEL
LIN {X 0,Y 285.338,Z 598.003,A -85,B 0,C 180,E1 -17203.17,E2 -17203.17} C_VEL
LIN {X 0,Y 286.683,Z 590.919,A -85,B 0,C 180,E1 -17205.28,E2 -17205.28} C_VEL
LIN {X 0,Y 288.494,Z 582.087,A -85,B 0,C 180,E1 -17207.363,E2 -17207.363} C_VEL
LIN {X 0,Y 290.081,Z 572.62,A -85,B 0,C 180,E1 -17209.168,E2 -17209.168} C_VEL
LIN {X 0,Y 291.576,Z 562.993,A -85,B 0,C 180,E1 -17210.642,E2 -17210.642} C_VEL
LIN {X 0,Y 293.292,Z 551.824,A -85,B 0,C 180,E1 -17211.988,E2 -17211.988} C_VEL
LIN {X 0,Y 294.818,Z 539.286,A -85,B 0,C 180,E1 -17213.163,E2 -17213.163} C_VEL
LIN {X 0,Y 296.012,Z 526.337,A -85,B 0,C 180,E1 -17214.038,E2 -17214.038} C_VEL
LIN {X 0,Y 296.886,Z 513.553,A -85,B 0,C 180,E1 -17214.613,E2 -17214.613} C_VEL
LIN {X 0,Y 297.84,Z 483.701,A -85,B 0,C 180,E1 -17215.363,E2 -17215.363} C_VEL
LIN {X 0,Y 298.897,Z 440.343,A -85,B 0,C 180,E1 -17216.401,E2 -17216.401} C_VEL
LIN {X 0,Y 297.317,Z 432.735,A -85,B 0,C 180,E1 -17216.755,E2 -17216.755} C_VEL
LIN {X 0,Y 290.18,Z 414.877,A -85,B 0,C 180,E1 -17217.962,E2 -17217.962} C_VEL
LIN {X 0,Y 285.909,Z 405.23,A -85,B 0,C 180,E1 -17218.721,E2 -17218.721} C_VEL
LIN {X 0,Y 284.347,Z 398.568,A -85,B 0,C 180,E1 -17221.424,E2 -17221.424} C_VEL
LIN {X 0,Y 284.344,Z 398.564,A -85,B 0,C 180,E1 -17225.348,E2 -17225.348} C_VEL
LIN {X 0,Y 284.315,Z 398.571,A -85,B 0,C 180,E1 -17228.169,E2 -17228.169} C_VEL
LIN {X 0,Y 284.273,Z 398.575,A -85,B 0,C 180,E1 -17232.125,E2 -17232.125} C_VEL
LIN {X 0,Y 284.289,Z 398.571,A -85,B 0,C 180,E1 -17236.195,E2 -17236.195} C_VEL
LIN {X 0,Y 284.355,Z 398.554,A -85,B 0,C 180,E1 -17240.013,E2 -17240.013} C_VEL
LIN {X 0,Y 284.355,Z 398.562,A -85,B 0,C 180,E1 -17243.617,E2 -17243.617} C_VEL
LIN {X 0,Y 284.312,Z 398.568,A -85,B 0,C 180,E1 -17247.19,E2 -17247.19} C_VEL
LIN {X 0,Y 284.363,Z 398.561,A -85,B 0,C 180,E1 -17250.376,E2 -17250.376} C_VEL
LIN {X 0,Y 284.397,Z 398.558,A -85,B 0,C 180,E1 -17252.786,E2 -17252.786} C_VEL
LIN {X 0,Y 284.143,Z 398.592,A -85,B 0,C 180,E1 -17253.576,E2 -17253.576} C_VEL
LIN {X 0,Y 282.811,Z 398.757,A -85,B 0,C 180,E1 -17254.741,E2 -17254.741} C_VEL
LIN {X 0,Y 278.404,Z 399.304,A -85,B 0,C 180,E1 -17257.45,E2 -17257.45} C_VEL
LIN {X 0,Y 277.376,Z 399.432,A -85,B 0,C 180,E1 -17258.662,E2 -17258.662} C_VEL
LIN {X 0,Y 277.318,Z 399.437,A -85,B 0,C 180,E1 -17259.073,E2 -17259.073} C_VEL
LIN {X 0,Y 277.366,Z 399.435,A -85,B 0,C 180,E1 -17262.298,E2 -17262.298} C_VEL
LIN {X 0,Y 277.439,Z 399.422,A -85,B 0,C 180,E1 -17265.326,E2 -17265.326} C_VEL
LIN {X 0,Y 277.511,Z 399.418,A -85,B 0,C 180,E1 -17269.789,E2 -17269.789} C_VEL
LIN {X 0,Y 277.658,Z 399.39,A -85,B 0,C 180,E1 -17272.729,E2 -17272.729} C_VEL
LIN {X 0,Y 277.825,Z 399.37,A -85,B 0,C 180,E1 -17278.55,E2 -17278.55} C_VEL
LIN {X 0,Y 277.825,Z 399.376,A -85,B 0,C 180,E1 -17281.449,E2 -17281.449} C_VEL
LIN {X 0,Y 277.634,Z 399.398,A -85,B 0,C 180,E1 -17287.271,E2 -17287.271} C_VEL
LIN {X 0,Y 277.465,Z 399.418,A -85,B 0,C 180,E1 -17290.213,E2 -17290.213} C_VEL
LIN {X 0,Y 277.439,Z 399.424,A -85,B 0,C 180,E1 -17294.674,E2 -17294.674} C_VEL
LIN {X 0,Y 277.349,Z 399.436,A -85,B 0,C 180,E1 -17299.234,E2 -17299.234} C_VEL
LIN {X 0,Y 277.323,Z 399.439,A -85,B 0,C 180,E1 -17304.17,E2 -17304.17} C_VEL
LIN {X 0,Y 277.327,Z 399.44,A -85,B 0,C 180,E1 -17307.504,E2 -17307.504} C_VEL
LIN {X 0,Y 277.275,Z 399.443,A -85,B 0,C 180,E1 -17310.481,E2 -17310.481} C_VEL
LIN {X 0,Y 277.25,Z 399.447,A -85,B 0,C 180,E1 -17313.895,E2 -17313.895} C_VEL
LIN {X 0,Y 277.268,Z 399.447,A -85,B 0,C 180,E1 -17317.469,E2 -17317.469} C_VEL
LIN {X 0,Y 277.213,Z 399.455,A -85,B 0,C 180,E1 -17321.236,E2 -17321.236} C_VEL
LIN {X 0,Y 277.219,Z 399.455,A -85,B 0,C 180,E1 -17325.223,E2 -17325.223} C_VEL
LIN {X 0,Y 277.225,Z 399.453,A -85,B 0,C 180,E1 -17329.512,E2 -17329.512} C_VEL
LIN {X 0,Y 277.27,Z 399.448,A -85,B 0,C 180,E1 -17332.531,E2 -17332.531} C_VEL
LIN {X 0,Y 277.325,Z 399.566,A -85,B 0,C 180,E1 -17334.403,E2 -17334.403} C_VEL
LIN {X 0,Y 279.574,Z 409.275,A -85,B 0,C 180,E1 -17338.136,E2 -17338.136} C_VEL
LIN {X 0,Y 281.114,Z 416.59,A -85,B 0,C 180,E1 -17340.808,E2 -17340.808} C_VEL
LIN {X 0,Y 287.215,Z 431.906,A -85,B 0,C 180,E1 -17341.909,E2 -17341.909} C_VEL
LIN {X 0,Y 291.009,Z 453.995,A -85,B 0,C 180,E1 -17342.905,E2 -17342.905} C_VEL
LIN {X 0,Y 292.061,Z 462.927,A -85,B 0,C 180,E1 -17343.251,E2 -17343.251} C_VEL
LIN {X 0,Y 290.193,Z 525,A -85,B 0,C 180,E1 -17344.78,E2 -17344.78} C_VEL
LIN {X 0,Y 289.173,Z 538.925,A -85,B 0,C 180,E1 -17345.404,E2 -17345.404} C_VEL
LIN {X 0,Y 287.862,Z 551.378,A -85,B 0,C 180,E1 -17346.244,E2 -17346.244} C_VEL
LIN {X 0,Y 286.348,Z 562.483,A -85,B 0,C 180,E1 -17347.259,E2 -17347.259} C_VEL
LIN {X 0,Y 284.748,Z 572.759,A -85,B 0,C 180,E1 -17348.46,E2 -17348.46} C_VEL
LIN {X 0,Y 282.802,Z 583.398,A -85,B 0,C 180,E1 -17350.019,E2 -17350.019} C_VEL
LIN {X 0,Y 280.955,Z 593.587,A -85,B 0,C 180,E1 -17351.908,E2 -17351.908} C_VEL
LIN {X 0,Y 279.378,Z 602.231,A -85,B 0,C 180,E1 -17353.935,E2 -17353.935} C_VEL
LIN {X 0,Y 277.874,Z 609.655,A -85,B 0,C 180,E1 -17356.097,E2 -17356.097} C_VEL
LIN {X 0,Y 276.757,Z 615.619,A -85,B 0,C 180,E1 -17358.278,E2 -17358.278} C_VEL
LIN {X 0,Y 275.993,Z 620.334,A -85,B 0,C 180,E1 -17360.472,E2 -17360.472} C_VEL
LIN {X 0,Y 275.497,Z 623.937,A -85,B 0,C 180,E1 -17362.672,E2 -17362.672} C_VEL
LIN {X 0,Y 275.224,Z 626.463,A -85,B 0,C 180,E1 -17364.804,E2 -17364.804} C_VEL
LIN {X 0,Y 275.242,Z 628.188,A -85,B 0,C 180,E1 -17367.072,E2 -17367.072} C_VEL
LIN {X 0,Y 275.248,Z 628.795,A -85,B 0,C 180,E1 -17368.537,E2 -17368.537} C_VEL
LIN {X 0,Y 275.246,Z 629.008,A -85,B 0,C 180,E1 -17370,E2 -17370} C_VEL
LIN {X 0,Y 275.248,Z 628.787,A -85,B 0,C 180,E1 -17371.463,E2 -17371.463} C_VEL
LIN {X 0,Y 275.242,Z 628.175,A -85,B 0,C 180,E1 -17372.927,E2 -17372.927} C_VEL
LIN {X 0,Y 275.237,Z 626.409,A -85,B 0,C 180,E1 -17375.227,E2 -17375.227} C_VEL
LIN {X 0,Y 275.617,Z 622.827,A -85,B 0,C 180,E1 -17378.062,E2 -17378.062} C_VEL
LIN {X 0,Y 276.207,Z 618.847,A -85,B 0,C 180,E1 -17380.26,E2 -17380.26} C_VEL
LIN {X 0,Y 277.214,Z 612.728,A -85,B 0,C 180,E1 -17382.816,E2 -17382.816} C_VEL
LIN {X 0,Y 278.597,Z 606.051,A -85,B 0,C 180,E1 -17384.985,E2 -17384.985} C_VEL
LIN {X 0,Y 280.22,Z 597.766,A -85,B 0,C 180,E1 -17387.139,E2 -17387.139} C_VEL
LIN {X 0,Y 281.728,Z 589.268,A -85,B 0,C 180,E1 -17388.923,E2 -17388.923} C_VEL
LIN {X 0,Y 283.611,Z 578.771,A -85,B 0,C 180,E1 -17390.678,E2 -17390.678} C_VEL
LIN {X 0,Y 285.597,Z 566.958,A -85,B 0,C 180,E1 -17392.231,E2 -17392.231} C_VEL
LIN {X 0,Y 287.308,Z 555.06,A -85,B 0,C 180,E1 -17393.422,E2 -17393.422} C_VEL
LIN {X 0,Y 288.675,Z 542.674,A -85,B 0,C 180,E1 -17394.353,E2 -17394.353} C_VEL
LIN {X 0,Y 289.892,Z 529.924,A -85,B 0,C 180,E1 -17395.008,E2 -17395.008} C_VEL
LIN {X 0,Y 290.519,Z 516.443,A -85,B 0,C 180,E1 -17395.429,E2 -17395.429} C_VEL
LIN {X 0,Y 291.929,Z 460.815,A -85,B 0,C 180,E1 -17396.788,E2 -17396.788} C_VEL
LIN {X 0,Y 288.127,Z 437.06,A -85,B 0,C 180,E1 -17397.82,E2 -17397.82} C_VEL
LIN {X 0,Y 286.883,Z 430.768,A -85,B 0,C 180,E1 -17398.125,E2 -17398.125} C_VEL
LIN {X 0,Y 281.106,Z 416.478,A -85,B 0,C 180,E1 -17399.192,E2 -17399.192} C_VEL
LIN {X 0,Y 279.022,Z 406.706,A -85,B 0,C 180,E1 -17402.789,E2 -17402.789} C_VEL
LIN {X 0,Y 277.285,Z 399.444,A -85,B 0,C 180,E1 -17405.658,E2 -17405.658} C_VEL
LIN {X 0,Y 277.235,Z 399.451,A -85,B 0,C 180,E1 -17409.328,E2 -17409.328} C_VEL
LIN {X 0,Y 277.217,Z 399.453,A -85,B 0,C 180,E1 -17413.196,E2 -17413.196} C_VEL
LIN {X 0,Y 277.219,Z 399.453,A -85,B 0,C 180,E1 -17417.324,E2 -17417.324} C_VEL
LIN {X 0,Y 277.263,Z 399.443,A -85,B 0,C 180,E1 -17421.793,E2 -17421.793} C_VEL
LIN {X 0,Y 277.285,Z 399.444,A -85,B 0,C 180,E1 -17424.341,E2 -17424.341} C_VEL
LIN {X 0,Y 277.245,Z 399.447,A -85,B 0,C 180,E1 -17427.836,E2 -17427.836} C_VEL
LIN {X 0,Y 277.269,Z 399.445,A -85,B 0,C 180,E1 -17431.21,E2 -17431.21} C_VEL
LIN {X 0,Y 277.314,Z 399.443,A -85,B 0,C 180,E1 -17434.48,E2 -17434.48} C_VEL
LIN {X 0,Y 277.293,Z 399.442,A -85,B 0,C 180,E1 -17437.655,E2 -17437.655} C_VEL
LIN {X 0,Y 277.347,Z 399.435,A -85,B 0,C 180,E1 -17440.766,E2 -17440.766} C_VEL
LIN {X 0,Y 277.437,Z 399.42,A -85,B 0,C 180,E1 -17445.326,E2 -17445.326} C_VEL
LIN {X 0,Y 277.462,Z 399.42,A -85,B 0,C 180,E1 -17449.787,E2 -17449.787} C_VEL
LIN {X 0,Y 277.631,Z 399.402,A -85,B 0,C 180,E1 -17452.729,E2 -17452.729} C_VEL
LIN {X 0,Y 277.823,Z 399.378,A -85,B 0,C 180,E1 -17458.551,E2 -17458.551} C_VEL
LIN {X 0,Y 277.824,Z 399.371,A -85,B 0,C 180,E1 -17461.45,E2 -17461.45} C_VEL
LIN {X 0,Y 277.656,Z 399.394,A -85,B 0,C 180,E1 -17467.271,E2 -17467.271} C_VEL
LIN {X 0,Y 277.508,Z 399.416,A -85,B 0,C 180,E1 -17470.211,E2 -17470.211} C_VEL
LIN {X 0,Y 277.436,Z 399.425,A -85,B 0,C 180,E1 -17474.674,E2 -17474.674} C_VEL
LIN {X 0,Y 277.349,Z 399.436,A -85,B 0,C 180,E1 -17479.234,E2 -17479.234} C_VEL
LIN {X 0,Y 277.331,Z 399.441,A -85,B 0,C 180,E1 -17483.92,E2 -17483.92} C_VEL
LIN {X 0,Y 277.328,Z 399.438,A -85,B 0,C 180,E1 -17487.506,E2 -17487.506} C_VEL
LIN {X 0,Y 277.273,Z 399.443,A -85,B 0,C 180,E1 -17490.481,E2 -17490.481} C_VEL
LIN {X 0,Y 277.256,Z 399.446,A -85,B 0,C 180,E1 -17493.895,E2 -17493.895} C_VEL
LIN {X 0,Y 277.285,Z 399.443,A -85,B 0,C 180,E1 -17497.467,E2 -17497.467} C_VEL
LIN {X 0,Y 277.234,Z 399.449,A -85,B 0,C 180,E1 -17501.232,E2 -17501.232} C_VEL
LIN {X 0,Y 277.202,Z 399.455,A -85,B 0,C 180,E1 -17505.227,E2 -17505.227} C_VEL
LIN {X 0,Y 277.224,Z 399.452,A -85,B 0,C 180,E1 -17509.512,E2 -17509.512} C_VEL
LIN {X 0,Y 277.269,Z 399.446,A -85,B 0,C 180,E1 -17512.531,E2 -17512.531} C_VEL
LIN {X 0,Y 277.249,Z 399.449,A -85,B 0,C 180,E1 -17516.105,E2 -17516.105} C_VEL
LIN {X 0,Y 277.263,Z 399.515,A -85,B 0,C 180,E1 -17518.148,E2 -17518.148} C_VEL
LIN {X 0,Y 278.662,Z 405.476,A -85,B 0,C 180,E1 -17520.606,E2 -17520.606} C_VEL
LIN {X 0,Y 286.198,Z 422.366,A -85,B 0,C 180,E1 -17521.944,E2 -17521.944} C_VEL
LIN {X 0,Y 291.492,Z 436.106,A -85,B 0,C 180,E1 -17522.876,E2 -17522.876} C_VEL
LIN {X 0,Y 292.557,Z 441.856,A -85,B 0,C 180,E1 -17523.139,E2 -17523.139} C_VEL
LIN {X 0,Y 290.542,Z 511.97,A -85,B 0,C 180,E1 -17524.861,E2 -17524.861} C_VEL
LIN {X 0,Y 289.642,Z 525.332,A -85,B 0,C 180,E1 -17525.448,E2 -17525.448} C_VEL
LIN {X 0,Y 288.415,Z 538.086,A -85,B 0,C 180,E1 -17526.293,E2 -17526.293} C_VEL
LIN {X 0,Y 287.011,Z 549.411,A -85,B 0,C 180,E1 -17527.315,E2 -17527.315} C_VEL
LIN {X 0,Y 285.294,Z 561.055,A -85,B 0,C 180,E1 -17528.694,E2 -17528.694} C_VEL
LIN {X 0,Y 283.523,Z 571.75,A -85,B 0,C 180,E1 -17530.304,E2 -17530.304} C_VEL
LIN {X 0,Y 282.13,Z 580.047,A -85,B 0,C 180,E1 -17531.858,E2 -17531.858} C_VEL
LIN {X 0,Y 280.55,Z 587.917,A -85,B 0,C 180,E1 -17533.631,E2 -17533.631} C_VEL
LIN {X 0,Y 278.892,Z 595.608,A -85,B 0,C 180,E1 -17535.777,E2 -17535.777} C_VEL
LIN {X 0,Y 277.463,Z 602.666,A -85,B 0,C 180,E1 -17538.309,E2 -17538.309} C_VEL
LIN {X 0,Y 276.529,Z 607.366,A -85,B 0,C 180,E1 -17540.491,E2 -17540.491} C_VEL
LIN {X 0,Y 275.932,Z 610.96,A -85,B 0,C 180,E1 -17542.684,E2 -17542.684} C_VEL
LIN {X 0,Y 275.659,Z 612.817,A -85,B 0,C 180,E1 -17544.147,E2 -17544.147} C_VEL
LIN {X 0,Y 275.511,Z 614.211,A -85,B 0,C 180,E1 -17545.611,E2 -17545.611} C_VEL
LIN {X 0,Y 275.406,Z 615.204,A -85,B 0,C 180,E1 -17547.075,E2 -17547.075} C_VEL
LIN {X 0,Y 275.252,Z 616.046,A -85,B 0,C 180,E1 -17550,E2 -17550} C_VEL
LIN {X 0,Y 275.29,Z 615.853,A -85,B 0,C 180,E1 -17551.463,E2 -17551.463} C_VEL
LIN {X 0,Y 275.405,Z 615.266,A -85,B 0,C 180,E1 -17552.926,E2 -17552.926} C_VEL
LIN {X 0,Y 275.508,Z 614.298,A -85,B 0,C 180,E1 -17554.389,E2 -17554.389} C_VEL
LIN {X 0,Y 275.736,Z 612.468,A -85,B 0,C 180,E1 -17556.257,E2 -17556.257} C_VEL
LIN {X 0,Y 276.312,Z 608.873,A -85,B 0,C 180,E1 -17558.779,E2 -17558.779} C_VEL
LIN {X 0,Y 277.091,Z 604.616,A -85,B 0,C 180,E1 -17560.966,E2 -17560.966} C_VEL
LIN {X 0,Y 278.433,Z 598.169,A -85,B 0,C 180,E1 -17563.502,E2 -17563.502} C_VEL
LIN {X 0,Y 279.843,Z 591.083,A -85,B 0,C 180,E1 -17565.663,E2 -17565.663} C_VEL
LIN {X 0,Y 281.733,Z 582.252,A -85,B 0,C 180,E1 -17567.794,E2 -17567.794} C_VEL
LIN {X 0,Y 283.327,Z 573.091,A -85,B 0,C 180,E1 -17569.585,E2 -17569.585} C_VEL
LIN {X 0,Y 284.965,Z 563.155,A -85,B 0,C 180,E1 -17571.143,E2 -17571.143} C_VEL
LIN {X 0,Y 286.72,Z 551.985,A -85,B 0,C 180,E1 -17572.52,E2 -17572.52} C_VEL
LIN {X 0,Y 288.325,Z 539.445,A -85,B 0,C 180,E1 -17573.716,E2 -17573.716} C_VEL
LIN {X 0,Y 289.567,Z 526.493,A -85,B 0,C 180,E1 -17574.608,E2 -17574.608} C_VEL
LIN {X 0,Y 290.463,Z 513.704,A -85,B 0,C 180,E1 -17575.195,E2 -17575.195} C_VEL
LIN {X 0,Y 291.404,Z 485.084,A -85,B 0,C 180,E1 -17575.931,E2 -17575.931} C_VEL
LIN {X 0,Y 292.572,Z 441.671,A -85,B 0,C 180,E1 -17576.986,E2 -17576.986} C_VEL
LIN {X 0,Y 291.142,Z 434.958,A -85,B 0,C 180,E1 -17577.313,E2 -17577.313} C_VEL
LIN {X 0,Y 284.243,Z 417.757,A -85,B 0,C 180,E1 -17578.522,E2 -17578.522} C_VEL
LIN {X 0,Y 278.701,Z 405.436,A -85,B 0,C 180,E1 -17579.528,E2 -17579.528} C_VEL
LIN {X 0,Y 277.298,Z 399.446,A -85,B 0,C 180,E1 -17582.056,E2 -17582.056} C_VEL
LIN {X 0,Y 277.284,Z 399.441,A -85,B 0,C 180,E1 -17585.799,E2 -17585.799} C_VEL
LIN {X 0,Y 277.237,Z 399.451,A -85,B 0,C 180,E1 -17589.328,E2 -17589.328} C_VEL
LIN {X 0,Y 277.22,Z 399.452,A -85,B 0,C 180,E1 -17593.197,E2 -17593.197} C_VEL
LIN {X 0,Y 277.241,Z 399.449,A -85,B 0,C 180,E1 -17597.32,E2 -17597.32} C_VEL
LIN {X 0,Y 277.268,Z 399.435,A -85,B 0,C 180,E1 -17600.677,E2 -17600.677} C_VEL
LIN {X 0,Y 277.324,Z 399.442,A -85,B 0,C 180,E1 -17604.347,E2 -17604.347} C_VEL
LIN {X 0,Y 277.249,Z 399.449,A -85,B 0,C 180,E1 -17607.837,E2 -17607.837} C_VEL
LIN {X 0,Y 277.293,Z 399.44,A -85,B 0,C 180,E1 -17611.213,E2 -17611.213} C_VEL
LIN {X 0,Y 277.318,Z 399.436,A -85,B 0,C 180,E1 -17614.48,E2 -17614.48} C_VEL
LIN {X 0,Y 277.297,Z 399.443,A -85,B 0,C 180,E1 -17617.656,E2 -17617.656} C_VEL
LIN {X 0,Y 277.318,Z 399.437,A -85,B 0,C 180,E1 -17619.073,E2 -17619.073} C_VEL
LIN {X 0,Y 276.733,Z 399.515,A -85,B 0,C 180,E1 -17620.286,E2 -17620.286} C_VEL
LIN {X 0,Y 273.95,Z 399.863,A -85,B 0,C 180,E1 -17622.263,E2 -17622.263} C_VEL
LIN {X 0,Y 271.529,Z 400.163,A -85,B 0,C 180,E1 -17623.87,E2 -17623.87} C_VEL
LIN {X 0,Y 270.465,Z 400.291,A -85,B 0,C 180,E1 -17625.114,E2 -17625.114} C_VEL
LIN {X 0,Y 270.367,Z 400.299,A -85,B 0,C 180,E1 -17625.536,E2 -17625.536} C_VEL
LIN {X 0,Y 270.446,Z 400.296,A -85,B 0,C 180,E1 -17629.519,E2 -17629.519} C_VEL
LIN {X 0,Y 270.616,Z 400.267,A -85,B 0,C 180,E1 -17632.539,E2 -17632.539} C_VEL
LIN {X 0,Y 270.791,Z 400.246,A -85,B 0,C 180,E1 -17638.513,E2 -17638.513} C_VEL
LIN {X 0,Y 270.791,Z 400.253,A -85,B 0,C 180,E1 -17641.487,E2 -17641.487} C_VEL
LIN {X 0,Y 270.59,Z 400.277,A -85,B 0,C 180,E1 -17647.462,E2 -17647.462} C_VEL
LIN {X 0,Y 270.417,Z 400.295,A -85,B 0,C 180,E1 -17650.482,E2 -17650.482} C_VEL
LIN {X 0,Y 270.407,Z 400.301,A -85,B 0,C 180,E1 -17655.064,E2 -17655.064} C_VEL
LIN {X 0,Y 270.305,Z 400.315,A -85,B 0,C 180,E1 -17659.755,E2 -17659.755} C_VEL
LIN {X 0,Y 270.278,Z 400.316,A -85,B 0,C 180,E1 -17664.585,E2 -17664.585} C_VEL
LIN {X 0,Y 270.273,Z 400.317,A -85,B 0,C 180,E1 -17667.908,E2 -17667.908} C_VEL
LIN {X 0,Y 270.187,Z 400.33,A -85,B 0,C 180,E1 -17671.348,E2 -17671.348} C_VEL
LIN {X 0,Y 270.204,Z 400.326,A -85,B 0,C 180,E1 -17674.905,E2 -17674.905} C_VEL
LIN {X 0,Y 270.2,Z 400.326,A -85,B 0,C 180,E1 -17678.71,E2 -17678.71} C_VEL
LIN {X 0,Y 270.174,Z 400.332,A -85,B 0,C 180,E1 -17683.25,E2 -17683.25} C_VEL
LIN {X 0,Y 270.177,Z 400.331,A -85,B 0,C 180,E1 -17687.442,E2 -17687.442} C_VEL
LIN {X 0,Y 270.209,Z 400.328,A -85,B 0,C 180,E1 -17691.374,E2 -17691.374} C_VEL
LIN {X 0,Y 270.232,Z 400.47,A -85,B 0,C 180,E1 -17693.729,E2 -17693.729} C_VEL
LIN {X 0,Y 272.325,Z 409.091,A -85,B 0,C 180,E1 -17697.183,E2 -17697.183} C_VEL
LIN {X 0,Y 273.919,Z 416.444,A -85,B 0,C 180,E1 -17699.966,E2 -17699.966} C_VEL
LIN {X 0,Y 281.192,Z 434.223,A -85,B 0,C 180,E1 -17701.322,E2 -17701.322} C_VEL
LIN {X 0,Y 285.331,Z 459.047,A -85,B 0,C 180,E1 -17702.464,E2 -17702.464} C_VEL
LIN {X 0,Y 285.705,Z 464.154,A -85,B 0,C 180,E1 -17702.644,E2 -17702.644} C_VEL
LIN {X 0,Y 283.795,Z 524.846,A -85,B 0,C 180,E1 -17704.17,E2 -17704.17} C_VEL
LIN {X 0,Y 282.744,Z 538.768,A -85,B 0,C 180,E1 -17704.807,E2 -17704.807} C_VEL
LIN {X 0,Y 281.382,Z 551.218,A -85,B 0,C 180,E1 -17705.662,E2 -17705.662} C_VEL
LIN {X 0,Y 279.809,Z 562.32,A -85,B 0,C 180,E1 -17706.696,E2 -17706.696} C_VEL
LIN {X 0,Y 277.918,Z 573.889,A -85,B 0,C 180,E1 -17708.099,E2 -17708.099} C_VEL
LIN {X 0,Y 275.94,Z 584.306,A -85,B 0,C 180,E1 -17709.694,E2 -17709.694} C_VEL
LIN {X 0,Y 274.05,Z 594.11,A -85,B 0,C 180,E1 -17711.598,E2 -17711.598} C_VEL
LIN {X 0,Y 272.513,Z 602.064,A -85,B 0,C 180,E1 -17713.519,E2 -17713.519} C_VEL
LIN {X 0,Y 270.98,Z 609.489,A -85,B 0,C 180,E1 -17715.736,E2 -17715.736} C_VEL
LIN {X 0,Y 269.754,Z 615.452,A -85,B 0,C 180,E1 -17717.969,E2 -17717.969} C_VEL
LIN {X 0,Y 268.972,Z 620.167,A -85,B 0,C 180,E1 -17720.221,E2 -17720.221} C_VEL
LIN {X 0,Y 268.422,Z 623.77,A -85,B 0,C 180,E1 -17722.477,E2 -17722.477} C_VEL
LIN {X 0,Y 268.124,Z 626.53,A -85,B 0,C 180,E1 -17724.906,E2 -17724.906} C_VEL
LIN {X 0,Y 268.153,Z 628.021,A -85,B 0,C 180,E1 -17726.995,E2 -17726.995} C_VEL
LIN {X 0,Y 268.174,Z 628.629,A -85,B 0,C 180,E1 -17728.498,E2 -17728.498} C_VEL
LIN {X 0,Y 268.171,Z 628.841,A -85,B 0,C 180,E1 -17730,E2 -17730} C_VEL
LIN {X 0,Y 268.174,Z 628.62,A -85,B 0,C 180,E1 -17731.501,E2 -17731.501} C_VEL
LIN {X 0,Y 268.153,Z 628.008,A -85,B 0,C 180,E1 -17733.004,E2 -17733.004} C_VEL
LIN {X 0,Y 268.163,Z 626.415,A -85,B 0,C 180,E1 -17735.187,E2 -17735.187} C_VEL
LIN {X 0,Y 268.564,Z 622.659,A -85,B 0,C 180,E1 -17738.275,E2 -17738.275} C_VEL
LIN {X 0,Y 269.207,Z 618.679,A -85,B 0,C 180,E1 -17740.529,E2 -17740.529} C_VEL
LIN {X 0,Y 270.275,Z 612.559,A -85,B 0,C 180,E1 -17743.151,E2 -17743.151} C_VEL
LIN {X 0,Y 271.735,Z 605.882,A -85,B 0,C 180,E1 -17745.373,E2 -17745.373} C_VEL
LIN {X 0,Y 273.428,Z 597.596,A -85,B 0,C 180,E1 -17747.578,E2 -17747.578} C_VEL
LIN {X 0,Y 274.985,Z 589.097,A -85,B 0,C 180,E1 -17749.405,E2 -17749.405} C_VEL
LIN {X 0,Y 276.967,Z 578.601,A -85,B 0,C 180,E1 -17751.198,E2 -17751.198} C_VEL
LIN {X 0,Y 279.047,Z 566.787,A -85,B 0,C 180,E1 -17752.782,E2 -17752.782} C_VEL
LIN {X 0,Y 280.815,Z 554.887,A -85,B 0,C 180,E1 -17753.997,E2 -17753.997} C_VEL
LIN {X 0,Y 282.226,Z 542.499,A -85,B 0,C 180,E1 -17754.947,E2 -17754.947} C_VEL
LIN {X 0,Y 283.489,Z 529.745,A -85,B 0,C 180,E1 -17755.613,E2 -17755.613} C_VEL
LIN {X 0,Y 284.141,Z 516.255,A -85,B 0,C 180,E1 -17756.042,E2 -17756.042} C_VEL
LIN {X 0,Y 285.528,Z 461.247,A -85,B 0,C 180,E1 -17757.421,E2 -17757.421} C_VEL
LIN {X 0,Y 281.391,Z 435.283,A -85,B 0,C 180,E1 -17758.591,E2 -17758.591} C_VEL
LIN {X 0,Y 280.081,Z 431.343,A -85,B 0,C 180,E1 -17758.849,E2 -17758.849} C_VEL
LIN {X 0,Y 273.882,Z 416.295,A -85,B 0,C 180,E1 -17760.038,E2 -17760.038} C_VEL
LIN {X 0,Y 271.91,Z 407.365,A -85,B 0,C 180,E1 -17763.451,E2 -17763.451} C_VEL
LIN {X 0,Y 270.232,Z 400.323,A -85,B 0,C 180,E1 -17766.353,E2 -17766.353} C_VEL
LIN {X 0,Y 270.175,Z 400.332,A -85,B 0,C 180,E1 -17770.566,E2 -17770.566} C_VEL
LIN {X 0,Y 270.166,Z 400.33,A -85,B 0,C 180,E1 -17774.617,E2 -17774.617} C_VEL
LIN {X 0,Y 270.17,Z 400.329,A -85,B 0,C 180,E1 -17778.972,E2 -17778.972} C_VEL
LIN {X 0,Y 270.217,Z 400.324,A -85,B 0,C 180,E1 -17783.259,E2 -17783.259} C_VEL
LIN {X 0,Y 270.204,Z 400.328,A -85,B 0,C 180,E1 -17786.893,E2 -17786.893} C_VEL
LIN {X 0,Y 270.196,Z 400.328,A -85,B 0,C 180,E1 -17790.383,E2 -17790.383} C_VEL
LIN {X 0,Y 270.264,Z 400.318,A -85,B 0,C 180,E1 -17793.764,E2 -17793.764} C_VEL
LIN {X 0,Y 270.238,Z 400.322,A -85,B 0,C 180,E1 -17797.039,E2 -17797.039} C_VEL
LIN {X 0,Y 270.304,Z 400.313,A -85,B 0,C 180,E1 -17800.245,E2 -17800.245} C_VEL
LIN {X 0,Y 270.405,Z 400.297,A -85,B 0,C 180,E1 -17804.935,E2 -17804.935} C_VEL
LIN {X 0,Y 270.414,Z 400.297,A -85,B 0,C 180,E1 -17809.518,E2 -17809.518} C_VEL
LIN {X 0,Y 270.587,Z 400.281,A -85,B 0,C 180,E1 -17812.538,E2 -17812.538} C_VEL
LIN {X 0,Y 270.788,Z 400.255,A -85,B 0,C 180,E1 -17818.513,E2 -17818.513} C_VEL
LIN {X 0,Y 270.79,Z 400.247,A -85,B 0,C 180,E1 -17821.487,E2 -17821.487} C_VEL
LIN {X 0,Y 270.614,Z 400.271,A -85,B 0,C 180,E1 -17827.461,E2 -17827.461} C_VEL
LIN {X 0,Y 270.443,Z 400.294,A -85,B 0,C 180,E1 -17830.481,E2 -17830.481} C_VEL
LIN {X 0,Y 270.405,Z 400.3,A -85,B 0,C 180,E1 -17835.065,E2 -17835.065} C_VEL
LIN {X 0,Y 270.305,Z 400.316,A -85,B 0,C 180,E1 -17839.755,E2 -17839.755} C_VEL
LIN {X 0,Y 270.276,Z 400.316,A -85,B 0,C 180,E1 -17844.586,E2 -17844.586} C_VEL
LIN {X 0,Y 270.273,Z 400.321,A -85,B 0,C 180,E1 -17847.909,E2 -17847.909} C_VEL
LIN {X 0,Y 270.186,Z 400.327,A -85,B 0,C 180,E1 -17851.348,E2 -17851.348} C_VEL
LIN {X 0,Y 270.225,Z 400.321,A -85,B 0,C 180,E1 -17854.902,E2 -17854.902} C_VEL
LIN {X 0,Y 270.223,Z 400.322,A -85,B 0,C 180,E1 -17858.717,E2 -17858.717} C_VEL
LIN {X 0,Y 270.181,Z 400.328,A -85,B 0,C 180,E1 -17862.557,E2 -17862.557} C_VEL
LIN {X 0,Y 270.166,Z 400.33,A -85,B 0,C 180,E1 -17866.751,E2 -17866.751} C_VEL
LIN {X 0,Y 270.175,Z 400.33,A -85,B 0,C 180,E1 -17869.434,E2 -17869.434} C_VEL
LIN {X 0,Y 270.228,Z 400.323,A -85,B 0,C 180,E1 -17873.731,E2 -17873.731} C_VEL
LIN {X 0,Y 270.236,Z 400.417,A -85,B 0,C 180,E1 -17877.507,E2 -17877.507} C_VEL
LIN {X 0,Y 271.466,Z 405.725,A -85,B 0,C 180,E1 -17879.762,E2 -17879.762} C_VEL
LIN {X 0,Y 280.1,Z 424.642,A -85,B 0,C 180,E1 -17881.337,E2 -17881.337} C_VEL
LIN {X 0,Y 285.445,Z 438.651,A -85,B 0,C 180,E1 -17882.318,E2 -17882.318} C_VEL
LIN {X 0,Y 286.231,Z 443.187,A -85,B 0,C 180,E1 -17882.527,E2 -17882.527} C_VEL
LIN {X 0,Y 284.151,Z 512.153,A -85,B 0,C 180,E1 -17884.254,E2 -17884.254} C_VEL
LIN {X 0,Y 283.204,Z 525.51,A -85,B 0,C 180,E1 -17884.851,E2 -17884.851} C_VEL
LIN {X 0,Y 281.935,Z 538.261,A -85,B 0,C 180,E1 -17885.713,E2 -17885.713} C_VEL
LIN {X 0,Y 280.484,Z 549.583,A -85,B 0,C 180,E1 -17886.756,E2 -17886.756} C_VEL
LIN {X 0,Y 278.713,Z 561.225,A -85,B 0,C 180,E1 -17888.165,E2 -17888.165} C_VEL
LIN {X 0,Y 276.782,Z 572.27,A -85,B 0,C 180,E1 -17889.867,E2 -17889.867} C_VEL
LIN {X 0,Y 275.06,Z 581.908,A -85,B 0,C 180,E1 -17891.76,E2 -17891.76} C_VEL
LIN {X 0,Y 273.075,Z 590.824,A -85,B 0,C 180,E1 -17893.939,E2 -17893.939} C_VEL
LIN {X 0,Y 271.58,Z 597.997,A -85,B 0,C 180,E1 -17896.151,E2 -17896.151} C_VEL
LIN {X 0,Y 270.514,Z 602.835,A -85,B 0,C 180,E1 -17898.004,E2 -17898.004} C_VEL
LIN {X 0,Y 269.53,Z 607.534,A -85,B 0,C 180,E1 -17900.242,E2 -17900.242} C_VEL
LIN {X 0,Y 268.892,Z 611.128,A -85,B 0,C 180,E1 -17902.491,E2 -17902.491} C_VEL
LIN {X 0,Y 268.588,Z 612.985,A -85,B 0,C 180,E1 -17903.992,E2 -17903.992} C_VEL
LIN {X 0,Y 268.422,Z 614.379,A -85,B 0,C 180,E1 -17905.495,E2 -17905.495} C_VEL
LIN {X 0,Y 268.319,Z 615.371,A -85,B 0,C 180,E1 -17906.997,E2 -17906.997} C_VEL
LIN {X 0,Y 268.178,Z 616.213,A -85,B 0,C 180,E1 -17910,E2 -17910} C_VEL
LIN {X 0,Y 268.219,Z 616.02,A -85,B 0,C 180,E1 -17911.502,E2 -17911.502} C_VEL
LIN {X 0,Y 268.318,Z 615.432,A -85,B 0,C 180,E1 -17913.003,E2 -17913.003} C_VEL
LIN {X 0,Y 268.419,Z 614.465,A -85,B 0,C 180,E1 -17914.505,E2 -17914.505} C_VEL
LIN {X 0,Y 268.616,Z 612.943,A -85,B 0,C 180,E1 -17916.16,E2 -17916.16} C_VEL
LIN {X 0,Y 269.28,Z 609.04,A -85,B 0,C 180,E1 -17919.01,E2 -17919.01} C_VEL
LIN {X 0,Y 270.123,Z 604.782,A -85,B 0,C 180,E1 -17921.253,E2 -17921.253} C_VEL
LIN {X 0,Y 271.525,Z 598.334,A -85,B 0,C 180,E1 -17923.853,E2 -17923.853} C_VEL
LIN {X 0,Y 273.015,Z 591.248,A -85,B 0,C 180,E1 -17926.065,E2 -17926.065} C_VEL
LIN {X 0,Y 274.969,Z 582.416,A -85,B 0,C 180,E1 -17928.247,E2 -17928.247} C_VEL
LIN {X 0,Y 276.768,Z 572.566,A -85,B 0,C 180,E1 -17930.202,E2 -17930.202} C_VEL
LIN {X 0,Y 278.366,Z 563.318,A -85,B 0,C 180,E1 -17931.669,E2 -17931.669} C_VEL
LIN {X 0,Y 280.179,Z 552.147,A -85,B 0,C 180,E1 -17933.076,E2 -17933.076} C_VEL
LIN {X 0,Y 281.865,Z 539.605,A -85,B 0,C 180,E1 -17934.294,E2 -17934.294} C_VEL
LIN {X 0,Y 283.147,Z 526.649,A -85,B 0,C 180,E1 -17935.204,E2 -17935.204} C_VEL
LIN {X 0,Y 284.08,Z 513.855,A -85,B 0,C 180,E1 -17935.802,E2 -17935.802} C_VEL
LIN {X 0,Y 284.899,Z 490.362,A -85,B 0,C 180,E1 -17936.427,E2 -17936.427} C_VEL
LIN {X 0,Y 286.231,Z 442.652,A -85,B 0,C 180,E1 -17937.611,E2 -17937.611} C_VEL
LIN {X 0,Y 285.041,Z 437.125,A -85,B 0,C 180,E1 -17937.891,E2 -17937.891} C_VEL
LIN {X 0,Y 277.346,Z 418.261,A -85,B 0,C 180,E1 -17939.289,E2 -17939.289} C_VEL
LIN {X 0,Y 271.484,Z 405.661,A -85,B 0,C 180,E1 -17940.38,E2 -17940.38} C_VEL
LIN {X 0,Y 270.211,Z 400.324,A -85,B 0,C 180,E1 -17942.719,E2 -17942.719} C_VEL
LIN {X 0,Y 270.221,Z 400.322,A -85,B 0,C 180,E1 -17946.741,E2 -17946.741} C_VEL
LIN {X 0,Y 270.172,Z 400.331,A -85,B 0,C 180,E1 -17951.029,E2 -17951.029} C_VEL
LIN {X 0,Y 270.175,Z 400.328,A -85,B 0,C 180,E1 -17955.384,E2 -17955.384} C_VEL
LIN {X 0,Y 270.216,Z 400.317,A -85,B 0,C 180,E1 -17959.441,E2 -17959.441} C_VEL
LIN {X 0,Y 270.259,Z 400.319,A -85,B 0,C 180,E1 -17963.722,E2 -17963.722} C_VEL
LIN {X 0,Y 270.208,Z 400.326,A -85,B 0,C 180,E1 -17966.893,E2 -17966.893} C_VEL
LIN {X 0,Y 270.233,Z 400.32,A -85,B 0,C 180,E1 -17970.387,E2 -17970.387} C_VEL
LIN {X 0,Y 270.268,Z 400.319,A -85,B 0,C 180,E1 -17973.764,E2 -17973.764} C_VEL
LIN {X 0,Y 270.242,Z 400.32,A -85,B 0,C 180,E1 -17977.039,E2 -17977.039} C_VEL
LIN {X 0,Y 270.307,Z 400.309,A -85,B 0,C 180,E1 -17980.245,E2 -17980.245} C_VEL
LIN {X 0,Y 270.407,Z 400.298,A -85,B 0,C 180,E1 -17984.935,E2 -17984.935} C_VEL
LIN {X 0,Y 270.367,Z 400.299,A -85,B 0,C 180,E1 -17985.536,E2 -17985.536} C_VEL
LIN {X 0,Y 269.684,Z 400.385,A -85,B 0,C 180,E1 -17986.78,E2 -17986.78} C_VEL
LIN {X 0,Y 266.892,Z 400.738,A -85,B 0,C 180,E1 -17988.809,E2 -17988.809} C_VEL
LIN {X 0,Y 264.573,Z 401.027,A -85,B 0,C 180,E1 -17990.458,E2 -17990.458} C_VEL
LIN {X 0,Y 263.622,Z 401.143,A -85,B 0,C 180,E1 -17991.735,E2 -17991.735} C_VEL
LIN {X 0,Y 263.567,Z 401.145,A -85,B 0,C 180,E1 -17992.167,E2 -17992.167} C_VEL
LIN {X 0,Y 263.569,Z 401.151,A -85,B 0,C 180,E1 -17996.943,E2 -17996.943} C_VEL
LIN {X 0,Y 263.808,Z 401.118,A -85,B 0,C 180,E1 -18000,E2 -18000} C_VEL
LIN {X 0,Y 263.568,Z 401.152,A -85,B 0,C 180,E1 -18003.057,E2 -18003.057} C_VEL
LIN {X 0,Y 263.549,Z 401.155,A -85,B 0,C 180,E1 -18007.662,E2 -18007.662} C_VEL
LIN {X 0,Y 263.359,Z 401.174,A -85,B 0,C 180,E1 -18010.766,E2 -18010.766} C_VEL
LIN {X 0,Y 263.355,Z 401.18,A -85,B 0,C 180,E1 -18015.478,E2 -18015.478} C_VEL
LIN {X 0,Y 263.267,Z 401.19,A -85,B 0,C 180,E1 -18020.306,E2 -18020.306} C_VEL
LIN {X 0,Y 263.212,Z 401.2,A -85,B 0,C 180,E1 -18025.291,E2 -18025.291} C_VEL
LIN {X 0,Y 263.169,Z 401.201,A -85,B 0,C 180,E1 -18028.731,E2 -18028.731} C_VEL
LIN {X 0,Y 263.136,Z 401.205,A -85,B 0,C 180,E1 -18032.288,E2 -18032.288} C_VEL
LIN {X 0,Y 263.185,Z 401.2,A -85,B 0,C 180,E1 -18036.763,E2 -18036.763} C_VEL
LIN {X 0,Y 263.128,Z 401.208,A -85,B 0,C 180,E1 -18041.593,E2 -18041.593} C_VEL
LIN {X 0,Y 263.13,Z 401.208,A -85,B 0,C 180,E1 -18046.017,E2 -18046.017} C_VEL
LIN {X 0,Y 263.108,Z 401.211,A -85,B 0,C 180,E1 -18050.127,E2 -18050.127} C_VEL
LIN {X 0,Y 263.172,Z 401.265,A -85,B 0,C 180,E1 -18052.975,E2 -18052.975} C_VEL
LIN {X 0,Y 265.591,Z 411.258,A -85,B 0,C 180,E1 -18057.111,E2 -18057.111} C_VEL
LIN {X 0,Y 266.712,Z 416.467,A -85,B 0,C 180,E1 -18059.073,E2 -18059.073} C_VEL
LIN {X 0,Y 274.714,Z 435.449,A -85,B 0,C 180,E1 -18060.62,E2 -18060.62} C_VEL
LIN {X 0,Y 275.621,Z 439.072,A -85,B 0,C 180,E1 -18060.832,E2 -18060.832} C_VEL
LIN {X 0,Y 279.118,Z 460.574,A -85,B 0,C 180,E1 -18061.845,E2 -18061.845} C_VEL
LIN {X 0,Y 279.391,Z 465.216,A -85,B 0,C 180,E1 -18062.007,E2 -18062.007} C_VEL
LIN {X 0,Y 277.421,Z 524.693,A -85,B 0,C 180,E1 -18063.531,E2 -18063.531} C_VEL
LIN {X 0,Y 276.352,Z 538.61,A -85,B 0,C 180,E1 -18064.182,E2 -18064.182} C_VEL
LIN {X 0,Y 274.917,Z 551.056,A -85,B 0,C 180,E1 -18065.051,E2 -18065.051} C_VEL
LIN {X 0,Y 273.295,Z 562.158,A -85,B 0,C 180,E1 -18066.107,E2 -18066.107} C_VEL
LIN {X 0,Y 271.346,Z 573.726,A -85,B 0,C 180,E1 -18067.54,E2 -18067.54} C_VEL
LIN {X 0,Y 269.257,Z 584.141,A -85,B 0,C 180,E1 -18069.167,E2 -18069.167} C_VEL
LIN {X 0,Y 267.573,Z 592.664,A -85,B 0,C 180,E1 -18070.833,E2 -18070.833} C_VEL
LIN {X 0,Y 265.987,Z 600.524,A -85,B 0,C 180,E1 -18072.707,E2 -18072.707} C_VEL
LIN {X 0,Y 264.317,Z 608.202,A -85,B 0,C 180,E1 -18074.974,E2 -18074.974} C_VEL
LIN {X 0,Y 262.765,Z 615.285,A -85,B 0,C 180,E1 -18077.644,E2 -18077.644} C_VEL
LIN {X 0,Y 261.949,Z 620.001,A -85,B 0,C 180,E1 -18079.956,E2 -18079.956} C_VEL
LIN {X 0,Y 261.357,Z 623.603,A -85,B 0,C 180,E1 -18082.273,E2 -18082.273} C_VEL
LIN {X 0,Y 261.024,Z 626.591,A -85,B 0,C 180,E1 -18085.015,E2 -18085.015} C_VEL
LIN {X 0,Y 261.048,Z 627.854,A -85,B 0,C 180,E1 -18086.913,E2 -18086.913} C_VEL
LIN {X 0,Y 261.08,Z 628.462,A -85,B 0,C 180,E1 -18088.457,E2 -18088.457} C_VEL
LIN {X 0,Y 261.098,Z 628.675,A -85,B 0,C 180,E1 -18090,E2 -18090} C_VEL
LIN {X 0,Y 261.08,Z 628.453,A -85,B 0,C 180,E1 -18091.542,E2 -18091.542} C_VEL
LIN {X 0,Y 261.048,Z 627.84,A -85,B 0,C 180,E1 -18093.086,E2 -18093.086} C_VEL
LIN {X 0,Y 261.085,Z 626.428,A -85,B 0,C 180,E1 -18095.137,E2 -18095.137} C_VEL
LIN {X 0,Y 261.357,Z 623.564,A -85,B 0,C 180,E1 -18097.727,E2 -18097.727} C_VEL
LIN {X 0,Y 261.948,Z 619.943,A -85,B 0,C 180,E1 -18100.043,E2 -18100.043} C_VEL
LIN {X 0,Y 262.756,Z 615.212,A -85,B 0,C 180,E1 -18102.355,E2 -18102.355} C_VEL
LIN {X 0,Y 264.302,Z 608.113,A -85,B 0,C 180,E1 -18105.026,E2 -18105.026} C_VEL
LIN {X 0,Y 265.979,Z 600.406,A -85,B 0,C 180,E1 -18107.293,E2 -18107.293} C_VEL
LIN {X 0,Y 267.918,Z 590.731,A -85,B 0,C 180,E1 -18109.539,E2 -18109.539} C_VEL
LIN {X 0,Y 269.885,Z 580.749,A -85,B 0,C 180,E1 -18111.381,E2 -18111.381} C_VEL
LIN {X 0,Y 271.984,Z 569.472,A -85,B 0,C 180,E1 -18113.006,E2 -18113.006} C_VEL
LIN {X 0,Y 273.799,Z 558.423,A -85,B 0,C 180,E1 -18114.248,E2 -18114.248} C_VEL
LIN {X 0,Y 275.438,Z 546.166,A -85,B 0,C 180,E1 -18115.302,E2 -18115.302} C_VEL
LIN {X 0,Y 276.709,Z 534.154,A -85,B 0,C 180,E1 -18116.035,E2 -18116.035} C_VEL
LIN {X 0,Y 277.61,Z 520.961,A -85,B 0,C 180,E1 -18116.55,E2 -18116.55} C_VEL
LIN {X 0,Y 279.236,Z 462.308,A -85,B 0,C 180,E1 -18118.058,E2 -18118.058} C_VEL
LIN {X 0,Y 275.217,Z 436.797,A -85,B 0,C 180,E1 -18119.244,E2 -18119.244} C_VEL
LIN {X 0,Y 268.121,Z 419.715,A -85,B 0,C 180,E1 -18120.609,E2 -18120.609} C_VEL
LIN {X 0,Y 266.622,Z 416.112,A -85,B 0,C 180,E1 -18120.938,E2 -18120.938} C_VEL
LIN {X 0,Y 264.573,Z 407.016,A -85,B 0,C 180,E1 -18124.566,E2 -18124.566} C_VEL
LIN {X 0,Y 263.171,Z 401.205,A -85,B 0,C 180,E1 -18127.025,E2 -18127.025} C_VEL
LIN {X 0,Y 263.126,Z 401.207,A -85,B 0,C 180,E1 -18131.594,E2 -18131.594} C_VEL
LIN {X 0,Y 263.129,Z 401.206,A -85,B 0,C 180,E1 -18136.017,E2 -18136.017} C_VEL
LIN {X 0,Y 263.106,Z 401.208,A -85,B 0,C 180,E1 -18140.128,E2 -18140.128} C_VEL
LIN {X 0,Y 263.163,Z 401.202,A -85,B 0,C 180,E1 -18144.018,E2 -18144.018} C_VEL
LIN {X 0,Y 263.134,Z 401.205,A -85,B 0,C 180,E1 -18147.712,E2 -18147.712} C_VEL
LIN {X 0,Y 263.197,Z 401.197,A -85,B 0,C 180,E1 -18151.785,E2 -18151.785} C_VEL
LIN {X 0,Y 263.227,Z 401.194,A -85,B 0,C 180,E1 -18155.2,E2 -18155.2} C_VEL
LIN {X 0,Y 263.27,Z 401.188,A -85,B 0,C 180,E1 -18159.694,E2 -18159.694} C_VEL
LIN {X 0,Y 263.353,Z 401.177,A -85,B 0,C 180,E1 -18164.522,E2 -18164.522} C_VEL
LIN {X 0,Y 263.357,Z 401.176,A -85,B 0,C 180,E1 -18169.234,E2 -18169.234} C_VEL
LIN {X 0,Y 263.546,Z 401.157,A -85,B 0,C 180,E1 -18172.338,E2 -18172.338} C_VEL
LIN {X 0,Y 263.753,Z 401.131,A -85,B 0,C 180,E1 -18178.473,E2 -18178.473} C_VEL
LIN {X 0,Y 263.754,Z 401.123,A -85,B 0,C 180,E1 -18181.527,E2 -18181.527} C_VEL
LIN {X 0,Y 263.575,Z 401.149,A -85,B 0,C 180,E1 -18187.662,E2 -18187.662} C_VEL
LIN {X 0,Y 263.376,Z 401.173,A -85,B 0,C 180,E1 -18190.766,E2 -18190.766} C_VEL
LIN {X 0,Y 263.353,Z 401.18,A -85,B 0,C 180,E1 -18195.478,E2 -18195.478} C_VEL
LIN {X 0,Y 263.271,Z 401.189,A -85,B 0,C 180,E1 -18200.306,E2 -18200.306} C_VEL
LIN {X 0,Y 263.21,Z 401.197,A -85,B 0,C 180,E1 -18205.291,E2 -18205.291} C_VEL
LIN {X 0,Y 263.181,Z 401.2,A -85,B 0,C 180,E1 -18208.73,E2 -18208.73} C_VEL
LIN {X 0,Y 263.135,Z 401.207,A -85,B 0,C 180,E1 -18212.288,E2 -18212.288} C_VEL
LIN {X 0,Y 263.192,Z 401.2,A -85,B 0,C 180,E1 -18215.978,E2 -18215.978} C_VEL
LIN {X 0,Y 263.139,Z 401.206,A -85,B 0,C 180,E1 -18219.867,E2 -18219.867} C_VEL
LIN {X 0,Y 263.124,Z 401.206,A -85,B 0,C 180,E1 -18223.984,E2 -18223.984} C_VEL
LIN {X 0,Y 263.125,Z 401.208,A -85,B 0,C 180,E1 -18228.407,E2 -18228.407} C_VEL
LIN {X 0,Y 263.184,Z 401.203,A -85,B 0,C 180,E1 -18233.237,E2 -18233.237} C_VEL
LIN {X 0,Y 263.173,Z 401.291,A -85,B 0,C 180,E1 -18236.808,E2 -18236.808} C_VEL
LIN {X 0,Y 264.294,Z 405.894,A -85,B 0,C 180,E1 -18238.849,E2 -18238.849} C_VEL
LIN {X 0,Y 273.735,Z 426.26,A -85,B 0,C 180,E1 -18240.649,E2 -18240.649} C_VEL
LIN {X 0,Y 279.423,Z 441.093,A -85,B 0,C 180,E1 -18241.733,E2 -18241.733} C_VEL
LIN {X 0,Y 279.872,Z 444.746,A -85,B 0,C 180,E1 -18241.887,E2 -18241.887} C_VEL
LIN {X 0,Y 277.794,Z 512.336,A -85,B 0,C 180,E1 -18243.62,E2 -18243.62} C_VEL
LIN {X 0,Y 276.811,Z 525.687,A -85,B 0,C 180,E1 -18244.228,E2 -18244.228} C_VEL
LIN {X 0,Y 275.779,Z 536.178,A -85,B 0,C 180,E1 -18244.933,E2 -18244.933} C_VEL
LIN {X 0,Y 274.262,Z 548.019,A -85,B 0,C 180,E1 -18245.996,E2 -18245.996} C_VEL
LIN {X 0,Y 272.563,Z 558.767,A -85,B 0,C 180,E1 -18247.246,E2 -18247.246} C_VEL
LIN {X 0,Y 270.655,Z 569.684,A -85,B 0,C 180,E1 -18248.876,E2 -18248.876} C_VEL
LIN {X 0,Y 268.958,Z 578.614,A -85,B 0,C 180,E1 -18250.539,E2 -18250.539} C_VEL
LIN {X 0,Y 266.957,Z 588.256,A -85,B 0,C 180,E1 -18252.772,E2 -18252.772} C_VEL
LIN {X 0,Y 265.111,Z 595.947,A -85,B 0,C 180,E1 -18255.021,E2 -18255.021} C_VEL
LIN {X 0,Y 263.577,Z 603.003,A -85,B 0,C 180,E1 -18257.684,E2 -18257.684} C_VEL
LIN {X 0,Y 262.522,Z 607.703,A -85,B 0,C 180,E1 -18259.979,E2 -18259.979} C_VEL
LIN {X 0,Y 261.849,Z 611.296,A -85,B 0,C 180,E1 -18262.288,E2 -18262.288} C_VEL
LIN {X 0,Y 261.501,Z 613.263,A -85,B 0,C 180,E1 -18263.935,E2 -18263.935} C_VEL
LIN {X 0,Y 261.234,Z 615.539,A -85,B 0,C 180,E1 -18266.916,E2 -18266.916} C_VEL
LIN {X 0,Y 261.149,Z 616.149,A -85,B 0,C 180,E1 -18268.458,E2 -18268.458} C_VEL
LIN {X 0,Y 261.105,Z 616.38,A -85,B 0,C 180,E1 -18270,E2 -18270} C_VEL
LIN {X 0,Y 261.149,Z 616.186,A -85,B 0,C 180,E1 -18271.542,E2 -18271.542} C_VEL
LIN {X 0,Y 261.233,Z 615.599,A -85,B 0,C 180,E1 -18273.085,E2 -18273.085} C_VEL
LIN {X 0,Y 261.518,Z 613.274,A -85,B 0,C 180,E1 -18276.171,E2 -18276.171} C_VEL
LIN {X 0,Y 262.051,Z 610.402,A -85,B 0,C 180,E1 -18278.483,E2 -18278.483} C_VEL
LIN {X 0,Y 262.826,Z 606.509,A -85,B 0,C 180,E1 -18280.789,E2 -18280.789} C_VEL
LIN {X 0,Y 263.898,Z 601.486,A -85,B 0,C 180,E1 -18283.084,E2 -18283.084} C_VEL
LIN {X 0,Y 265.306,Z 595.158,A -85,B 0,C 180,E1 -18285.361,E2 -18285.361} C_VEL
LIN {X 0,Y 267.161,Z 587.237,A -85,B 0,C 180,E1 -18287.61,E2 -18287.61} C_VEL
LIN {X 0,Y 268.858,Z 579.164,A -85,B 0,C 180,E1 -18289.469,E2 -18289.469} C_VEL
LIN {X 0,Y 270.698,Z 569.313,A -85,B 0,C 180,E1 -18291.314,E2 -18291.314} C_VEL
LIN {X 0,Y 272.72,Z 558.218,A -85,B 0,C 180,E1 -18292.941,E2 -18292.941} C_VEL
LIN {X 0,Y 274.42,Z 547.341,A -85,B 0,C 180,E1 -18294.191,E2 -18294.191} C_VEL
LIN {X 0,Y 275.923,Z 535.319,A -85,B 0,C 180,E1 -18295.255,E2 -18295.255} C_VEL
LIN {X 0,Y 277.098,Z 522.952,A -85,B 0,C 180,E1 -18296.047,E2 -18296.047} C_VEL
LIN {X 0,Y 277.917,Z 510.108,A -85,B 0,C 180,E1 -18296.57,E2 -18296.57} C_VEL
LIN {X 0,Y 278.877,Z 479.503,A -85,B 0,C 180,E1 -18297.356,E2 -18297.356} C_VEL
LIN {X 0,Y 279.953,Z 443.669,A -85,B 0,C 180,E1 -18298.26,E2 -18298.26} C_VEL
LIN {X 0,Y 278.819,Z 439.119,A -85,B 0,C 180,E1 -18298.517,E2 -18298.517} C_VEL
LIN {X 0,Y 271.851,Z 421.866,A -85,B 0,C 180,E1 -18299.837,E2 -18299.837} C_VEL
LIN {X 0,Y 264.289,Z 405.847,A -85,B 0,C 180,E1 -18301.299,E2 -18301.299} C_VEL
LIN {X 0,Y 263.167,Z 401.201,A -85,B 0,C 180,E1 -18303.423,E2 -18303.423} C_VEL
LIN {X 0,Y 263.162,Z 401.205,A -85,B 0,C 180,E1 -18307.897,E2 -18307.897} C_VEL
LIN {X 0,Y 263.128,Z 401.208,A -85,B 0,C 180,E1 -18311.893,E2 -18311.893} C_VEL
LIN {X 0,Y 263.138,Z 401.205,A -85,B 0,C 180,E1 -18316.148,E2 -18316.148} C_VEL
LIN {X 0,Y 263.142,Z 401.192,A -85,B 0,C 180,E1 -18320.134,E2 -18320.134} C_VEL
LIN {X 0,Y 263.194,Z 401.2,A -85,B 0,C 180,E1 -18324.023,E2 -18324.023} C_VEL
LIN {X 0,Y 263.137,Z 401.206,A -85,B 0,C 180,E1 -18327.712,E2 -18327.712} C_VEL
LIN {X 0,Y 263.205,Z 401.196,A -85,B 0,C 180,E1 -18331.783,E2 -18331.783} C_VEL
LIN {X 0,Y 263.23,Z 401.188,A -85,B 0,C 180,E1 -18335.2,E2 -18335.2} C_VEL
LIN {X 0,Y 263.273,Z 401.188,A -85,B 0,C 180,E1 -18339.694,E2 -18339.694} C_VEL
LIN {X 0,Y 263.355,Z 401.178,A -85,B 0,C 180,E1 -18344.522,E2 -18344.522} C_VEL
LIN {X 0,Y 263.378,Z 401.176,A -85,B 0,C 180,E1 -18349.234,E2 -18349.234} C_VEL
LIN {X 0,Y 263.567,Z 401.145,A -85,B 0,C 180,E1 -18352.167,E2 -18352.167} C_VEL
LIN {X 0,Y 262.969,Z 401.223,A -85,B 0,C 180,E1 -18353.44,E2 -18353.44} C_VEL
LIN {X 0,Y 260.19,Z 401.574,A -85,B 0,C 180,E1 -18355.518,E2 -18355.518} C_VEL
LIN {X 0,Y 257.804,Z 401.87,A -85,B 0,C 180,E1 -18357.207,E2 -18357.207} C_VEL
LIN {X 0,Y 256.79,Z 401.989,A -85,B 0,C 180,E1 -18358.517,E2 -18358.517} C_VEL
LIN {X 0,Y 256.714,Z 401.997,A -85,B 0,C 180,E1 -18358.96,E2 -18358.96} C_VEL
LIN {X 0,Y 256.718,Z 402.006,A -85,B 0,C 180,E1 -18361.569,E2 -18361.569} C_VEL
LIN {X 0,Y 256.48,Z 402.032,A -85,B 0,C 180,E1 -18366.293,E2 -18366.293} C_VEL
LIN {X 0,Y 256.43,Z 402.044,A -85,B 0,C 180,E1 -18369.465,E2 -18369.465} C_VEL
LIN {X 0,Y 256.261,Z 402.063,A -85,B 0,C 180,E1 -18374.29,E2 -18374.29} C_VEL
LIN {X 0,Y 256.215,Z 402.064,A -85,B 0,C 180,E1 -18377.562,E2 -18377.562} C_VEL
LIN {X 0,Y 256.162,Z 402.076,A -85,B 0,C 180,E1 -18381.12,E2 -18381.12} C_VEL
LIN {X 0,Y 256.192,Z 402.074,A -85,B 0,C 180,E1 -18385.138,E2 -18385.138} C_VEL
LIN {X 0,Y 256.107,Z 402.083,A -85,B 0,C 180,E1 -18389.601,E2 -18389.601} C_VEL
LIN {X 0,Y 256.071,Z 402.088,A -85,B 0,C 180,E1 -18393.292,E2 -18393.292} C_VEL
LIN {X 0,Y 256.117,Z 402.082,A -85,B 0,C 180,E1 -18397.27,E2 -18397.27} C_VEL
LIN {X 0,Y 256.058,Z 402.09,A -85,B 0,C 180,E1 -18401.203,E2 -18401.203} C_VEL
LIN {X 0,Y 256.065,Z 402.09,A -85,B 0,C 180,E1 -18405.529,E2 -18405.529} C_VEL
LIN {X 0,Y 256.058,Z 402.091,A -85,B 0,C 180,E1 -18408.796,E2 -18408.796} C_VEL
LIN {X 0,Y 256.148,Z 402.229,A -85,B 0,C 180,E1 -18412.248,E2 -18412.248} C_VEL
LIN {X 0,Y 258.319,Z 411.166,A -85,B 0,C 180,E1 -18416.1,E2 -18416.1} C_VEL
LIN {X 0,Y 259.466,Z 416.281,A -85,B 0,C 180,E1 -18418.109,E2 -18418.109} C_VEL
LIN {X 0,Y 266.935,Z 433.396,A -85,B 0,C 180,E1 -18419.619,E2 -18419.619} C_VEL
LIN {X 0,Y 269.341,Z 439.708,A -85,B 0,C 180,E1 -18420.107,E2 -18420.107} C_VEL
LIN {X 0,Y 272.451,Z 458.961,A -85,B 0,C 180,E1 -18421.049,E2 -18421.049} C_VEL
LIN {X 0,Y 273.135,Z 464.879,A -85,B 0,C 180,E1 -18421.301,E2 -18421.301} C_VEL
LIN {X 0,Y 271.105,Z 524.54,A -85,B 0,C 180,E1 -18422.864,E2 -18422.864} C_VEL
LIN {X 0,Y 269.961,Z 538.451,A -85,B 0,C 180,E1 -18423.524,E2 -18423.524} C_VEL
LIN {X 0,Y 268.5,Z 550.896,A -85,B 0,C 180,E1 -18424.412,E2 -18424.412} C_VEL
LIN {X 0,Y 266.798,Z 561.995,A -85,B 0,C 180,E1 -18425.487,E2 -18425.487} C_VEL
LIN {X 0,Y 264.79,Z 573.562,A -85,B 0,C 180,E1 -18426.952,E2 -18426.952} C_VEL
LIN {X 0,Y 262.62,Z 583.977,A -85,B 0,C 180,E1 -18428.615,E2 -18428.615} C_VEL
LIN {X 0,Y 260.767,Z 592.848,A -85,B 0,C 180,E1 -18430.394,E2 -18430.394} C_VEL
LIN {X 0,Y 258.864,Z 601.733,A -85,B 0,C 180,E1 -18432.623,E2 -18432.623} C_VEL
LIN {X 0,Y 257.174,Z 609.156,A -85,B 0,C 180,E1 -18434.952,E2 -18434.952} C_VEL
LIN {X 0,Y 255.791,Z 615.118,A -85,B 0,C 180,E1 -18437.302,E2 -18437.302} C_VEL
LIN {X 0,Y 254.917,Z 619.834,A -85,B 0,C 180,E1 -18439.676,E2 -18439.676} C_VEL
LIN {X 0,Y 254.317,Z 623.437,A -85,B 0,C 180,E1 -18442.057,E2 -18442.057} C_VEL
LIN {X 0,Y 254.065,Z 625.295,A -85,B 0,C 180,E1 -18443.647,E2 -18443.647} C_VEL
LIN {X 0,Y 253.954,Z 626.689,A -85,B 0,C 180,E1 -18445.237,E2 -18445.237} C_VEL
LIN {X 0,Y 253.948,Z 627.686,A -85,B 0,C 180,E1 -18446.827,E2 -18446.827} C_VEL
LIN {X 0,Y 253.988,Z 628.295,A -85,B 0,C 180,E1 -18448.414,E2 -18448.414} C_VEL
LIN {X 0,Y 254.027,Z 628.508,A -85,B 0,C 180,E1 -18450,E2 -18450} C_VEL
LIN {X 0,Y 253.988,Z 628.286,A -85,B 0,C 180,E1 -18451.585,E2 -18451.585} C_VEL
LIN {X 0,Y 253.948,Z 627.672,A -85,B 0,C 180,E1 -18453.173,E2 -18453.173} C_VEL
LIN {X 0,Y 253.99,Z 626.47,A -85,B 0,C 180,E1 -18455.039,E2 -18455.039} C_VEL
LIN {X 0,Y 254.316,Z 623.396,A -85,B 0,C 180,E1 -18457.942,E2 -18457.942} C_VEL
LIN {X 0,Y 254.916,Z 619.774,A -85,B 0,C 180,E1 -18460.323,E2 -18460.323} C_VEL
LIN {X 0,Y 255.783,Z 615.042,A -85,B 0,C 180,E1 -18462.698,E2 -18462.698} C_VEL
LIN {X 0,Y 257.438,Z 607.944,A -85,B 0,C 180,E1 -18465.436,E2 -18465.436} C_VEL
LIN {X 0,Y 259.191,Z 600.264,A -85,B 0,C 180,E1 -18467.753,E2 -18467.753} C_VEL
LIN {X 0,Y 261.212,Z 590.56,A -85,B 0,C 180,E1 -18470.062,E2 -18470.062} C_VEL
LIN {X 0,Y 263.268,Z 580.578,A -85,B 0,C 180,E1 -18471.946,E2 -18471.946} C_VEL
LIN {X 0,Y 265.457,Z 569.3,A -85,B 0,C 180,E1 -18473.605,E2 -18473.605} C_VEL
LIN {X 0,Y 267.33,Z 558.25,A -85,B 0,C 180,E1 -18474.874,E2 -18474.874} C_VEL
LIN {X 0,Y 269.017,Z 545.991,A -85,B 0,C 180,E1 -18475.95,E2 -18475.95} C_VEL
LIN {X 0,Y 270.427,Z 533.06,A -85,B 0,C 180,E1 -18476.739,E2 -18476.739} C_VEL
LIN {X 0,Y 271.353,Z 519.271,A -85,B 0,C 180,E1 -18477.265,E2 -18477.265} C_VEL
LIN {X 0,Y 272.983,Z 463.333,A -85,B 0,C 180,E1 -18478.724,E2 -18478.724} C_VEL
LIN {X 0,Y 269.684,Z 442.072,A -85,B 0,C 180,E1 -18479.741,E2 -18479.741} C_VEL
LIN {X 0,Y 268.839,Z 438.18,A -85,B 0,C 180,E1 -18479.961,E2 -18479.961} C_VEL
LIN {X 0,Y 262.043,Z 422.11,A -85,B 0,C 180,E1 -18481.317,E2 -18481.317} C_VEL
LIN {X 0,Y 259.395,Z 415.988,A -85,B 0,C 180,E1 -18481.877,E2 -18481.877} C_VEL
LIN {X 0,Y 257.154,Z 406.127,A -85,B 0,C 180,E1 -18485.985,E2 -18485.985} C_VEL
LIN {X 0,Y 256.129,Z 402.079,A -85,B 0,C 180,E1 -18487.818,E2 -18487.818} C_VEL
LIN {X 0,Y 256.074,Z 402.085,A -85,B 0,C 180,E1 -18492.181,E2 -18492.181} C_VEL
LIN {X 0,Y 256.065,Z 402.085,A -85,B 0,C 180,E1 -18496.674,E2 -18496.674} C_VEL
LIN {X 0,Y 256.072,Z 402.087,A -85,B 0,C 180,E1 -18500.858,E2 -18500.858} C_VEL
LIN {X 0,Y 256.131,Z 402.078,A -85,B 0,C 180,E1 -18502.867,E2 -18502.867} C_VEL
LIN {X 0,Y 256.068,Z 402.088,A -85,B 0,C 180,E1 -18506.707,E2 -18506.707} C_VEL
LIN {X 0,Y 256.104,Z 402.084,A -85,B 0,C 180,E1 -18510.399,E2 -18510.399} C_VEL
LIN {X 0,Y 256.189,Z 402.072,A -85,B 0,C 180,E1 -18514.861,E2 -18514.861} C_VEL
LIN {X 0,Y 256.219,Z 402.067,A -85,B 0,C 180,E1 -18519.109,E2 -18519.109} C_VEL
LIN {X 0,Y 256.302,Z 402.059,A -85,B 0,C 180,E1 -18524.085,E2 -18524.085} C_VEL
LIN {X 0,Y 256.298,Z 402.058,A -85,B 0,C 180,E1 -18527.328,E2 -18527.328} C_VEL
LIN {X 0,Y 256.506,Z 402.032,A -85,B 0,C 180,E1 -18532.126,E2 -18532.126} C_VEL
LIN {X 0,Y 256.5,Z 402.032,A -85,B 0,C 180,E1 -18536.859,E2 -18536.859} C_VEL
LIN {X 0,Y 256.767,Z 401.998,A -85,B 0,C 180,E1 -18540,E2 -18540} C_VEL
LIN {X 0,Y 256.503,Z 402.032,A -85,B 0,C 180,E1 -18543.141,E2 -18543.141} C_VEL
LIN {X 0,Y 256.542,Z 402.026,A -85,B 0,C 180,E1 -18547.873,E2 -18547.873} C_VEL
LIN {X 0,Y 256.311,Z 402.053,A -85,B 0,C 180,E1 -18551.066,E2 -18551.066} C_VEL
LIN {X 0,Y 256.302,Z 402.056,A -85,B 0,C 180,E1 -18555.915,E2 -18555.915} C_VEL
LIN {X 0,Y 256.22,Z 402.065,A -85,B 0,C 180,E1 -18560.891,E2 -18560.891} C_VEL
LIN {X 0,Y 256.19,Z 402.071,A -85,B 0,C 180,E1 -18565.139,E2 -18565.139} C_VEL
LIN {X 0,Y 256.115,Z 402.081,A -85,B 0,C 180,E1 -18569.6,E2 -18569.6} C_VEL
LIN {X 0,Y 256.087,Z 402.086,A -85,B 0,C 180,E1 -18573.29,E2 -18573.29} C_VEL
LIN {X 0,Y 256.141,Z 402.077,A -85,B 0,C 180,E1 -18577.278,E2 -18577.278} C_VEL
LIN {X 0,Y 256.073,Z 402.084,A -85,B 0,C 180,E1 -18581.2,E2 -18581.2} C_VEL
LIN {X 0,Y 256.046,Z 402.093,A -85,B 0,C 180,E1 -18585.533,E2 -18585.533} C_VEL
LIN {X 0,Y 256.056,Z 402.09,A -85,B 0,C 180,E1 -18588.797,E2 -18588.797} C_VEL
LIN {X 0,Y 256.132,Z 402.081,A -85,B 0,C 180,E1 -18592.868,E2 -18592.868} C_VEL
LIN {X 0,Y 256.138,Z 402.154,A -85,B 0,C 180,E1 -18596.06,E2 -18596.06} C_VEL
LIN {X 0,Y 257.051,Z 406.085,A -85,B 0,C 180,E1 -18597.867,E2 -18597.867} C_VEL
LIN {X 0,Y 266.759,Z 426.535,A -85,B 0,C 180,E1 -18599.804,E2 -18599.804} C_VEL
LIN {X 0,Y 273.257,Z 442.899,A -85,B 0,C 180,E1 -18601.083,E2 -18601.083} C_VEL
LIN {X 0,Y 273.61,Z 445.849,A -85,B 0,C 180,E1 -18601.211,E2 -18601.211} C_VEL
LIN {X 0,Y 271.449,Z 512.52,A -85,B 0,C 180,E1 -18602.954,E2 -18602.954} C_VEL
LIN {X 0,Y 270.455,Z 525.863,A -85,B 0,C 180,E1 -18603.576,E2 -18603.576} C_VEL
LIN {X 0,Y 269.354,Z 536.353,A -85,B 0,C 180,E1 -18604.292,E2 -18604.292} C_VEL
LIN {X 0,Y 267.809,Z 548.192,A -85,B 0,C 180,E1 -18605.38,E2 -18605.38} C_VEL
LIN {X 0,Y 266.048,Z 558.938,A -85,B 0,C 180,E1 -18606.657,E2 -18606.657} C_VEL
LIN {X 0,Y 264.265,Z 568.815,A -85,B 0,C 180,E1 -18608.141,E2 -18608.141} C_VEL
LIN {X 0,Y 262.262,Z 578.784,A -85,B 0,C 180,E1 -18610.022,E2 -18610.022} C_VEL
LIN {X 0,Y 260.485,Z 586.947,A -85,B 0,C 180,E1 -18611.924,E2 -18611.924} C_VEL
LIN {X 0,Y 258.514,Z 594.948,A -85,B 0,C 180,E1 -18614.225,E2 -18614.225} C_VEL
LIN {X 0,Y 257.04,Z 601.364,A -85,B 0,C 180,E1 -18616.561,E2 -18616.561} C_VEL
LIN {X 0,Y 255.854,Z 606.454,A -85,B 0,C 180,E1 -18618.914,E2 -18618.914} C_VEL
LIN {X 0,Y 255.019,Z 610.404,A -85,B 0,C 180,E1 -18621.282,E2 -18621.282} C_VEL
LIN {X 0,Y 254.385,Z 613.68,A -85,B 0,C 180,E1 -18624.039,E2 -18624.039} C_VEL
LIN {X 0,Y 254.152,Z 615.706,A -85,B 0,C 180,E1 -18626.83,E2 -18626.83} C_VEL
LIN {X 0,Y 254.034,Z 616.546,A -85,B 0,C 180,E1 -18630,E2 -18630} C_VEL
LIN {X 0,Y 254.058,Z 616.353,A -85,B 0,C 180,E1 -18631.585,E2 -18631.585} C_VEL
LIN {X 0,Y 254.151,Z 615.766,A -85,B 0,C 180,E1 -18633.171,E2 -18633.171} C_VEL
LIN {X 0,Y 254.455,Z 613.44,A -85,B 0,C 180,E1 -18636.343,E2 -18636.343} C_VEL
LIN {X 0,Y 255.029,Z 610.569,A -85,B 0,C 180,E1 -18638.718,E2 -18638.718} C_VEL
LIN {X 0,Y 255.833,Z 606.675,A -85,B 0,C 180,E1 -18641.087,E2 -18641.087} C_VEL
LIN {X 0,Y 256.975,Z 601.651,A -85,B 0,C 180,E1 -18643.443,E2 -18643.443} C_VEL
LIN {X 0,Y 258.469,Z 595.323,A -85,B 0,C 180,E1 -18645.778,E2 -18645.778} C_VEL
LIN {X 0,Y 260.407,Z 587.401,A -85,B 0,C 180,E1 -18648.082,E2 -18648.082} C_VEL
LIN {X 0,Y 262.34,Z 578.511,A -85,B 0,C 180,E1 -18650.161,E2 -18650.161} C_VEL
LIN {X 0,Y 264.291,Z 568.378,A -85,B 0,C 180,E1 -18652.063,E2 -18652.063} C_VEL
LIN {X 0,Y 266.441,Z 556.958,A -85,B 0,C 180,E1 -18653.72,E2 -18653.72} C_VEL
LIN {X 0,Y 268.26,Z 545.739,A -85,B 0,C 180,E1 -18654.99,E2 -18654.99} C_VEL
LIN {X 0,Y 269.682,Z 534.342,A -85,B 0,C 180,E1 -18655.986,E2 -18655.986} C_VEL
LIN {X 0,Y 270.883,Z 521.287,A -85,B 0,C 180,E1 -18656.795,E2 -18656.795} C_VEL
LIN {X 0,Y 271.648,Z 508.75,A -85,B 0,C 180,E1 -18657.285,E2 -18657.285} C_VEL
LIN {X 0,Y 272.503,Z 483.248,A -85,B 0,C 180,E1 -18657.946,E2 -18657.946} C_VEL
LIN {X 0,Y 273.634,Z 444.522,A -85,B 0,C 180,E1 -18658.953,E2 -18658.953} C_VEL
LIN {X 0,Y 272.467,Z 440.688,A -85,B 0,C 180,E1 -18659.203,E2 -18659.203} C_VEL
LIN {X 0,Y 265.729,Z 424.132,A -85,B 0,C 180,E1 -18660.531,E2 -18660.531} C_VEL
LIN {X 0,Y 258.468,Z 409.123,A -85,B 0,C 180,E1 -18661.972,E2 -18661.972} C_VEL
LIN {X 0,Y 257.078,Z 406.058,A -85,B 0,C 180,E1 -18662.272,E2 -18662.272} C_VEL
LIN {X 0,Y 256.135,Z 402.082,A -85,B 0,C 180,E1 -18664.162,E2 -18664.162} C_VEL
LIN {X 0,Y 256.118,Z 402.082,A -85,B 0,C 180,E1 -18667.271,E2 -18667.271} C_VEL
LIN {X 0,Y 256.058,Z 402.089,A -85,B 0,C 180,E1 -18671.203,E2 -18671.203} C_VEL
LIN {X 0,Y 256.069,Z 402.085,A -85,B 0,C 180,E1 -18675.528,E2 -18675.528} C_VEL
LIN {X 0,Y 256.079,Z 402.079,A -85,B 0,C 180,E1 -18678.801,E2 -18678.801} C_VEL
LIN {X 0,Y 256.157,Z 402.076,A -85,B 0,C 180,E1 -18682.872,E2 -18682.872} C_VEL
LIN {X 0,Y 256.089,Z 402.084,A -85,B 0,C 180,E1 -18686.71,E2 -18686.71} C_VEL
LIN {X 0,Y 256.142,Z 402.075,A -85,B 0,C 180,E1 -18691.405,E2 -18691.405} C_VEL
LIN {X 0,Y 256.172,Z 402.067,A -85,B 0,C 180,E1 -18695.699,E2 -18695.699} C_VEL
LIN {X 0,Y 256.223,Z 402.066,A -85,B 0,C 180,E1 -18699.11,E2 -18699.11} C_VEL
LIN {X 0,Y 256.304,Z 402.059,A -85,B 0,C 180,E1 -18704.085,E2 -18704.085} C_VEL
LIN {X 0,Y 256.314,Z 402.056,A -85,B 0,C 180,E1 -18708.934,E2 -18708.934} C_VEL
LIN {X 0,Y 256.544,Z 402.02,A -85,B 0,C 180,E1 -18712.134,E2 -18712.134} C_VEL
LIN {X 0,Y 256.719,Z 401.998,A -85,B 0,C 180,E1 -18718.431,E2 -18718.431} C_VEL
LIN {X 0,Y 256.714,Z 401.997,A -85,B 0,C 180,E1 -18718.96,E2 -18718.96} C_VEL
LIN {X 0,Y 256.387,Z 402.041,A -85,B 0,C 180,E1 -18719.835,E2 -18719.835} C_VEL
LIN {X 0,Y 254.957,Z 402.224,A -85,B 0,C 180,E1 -18721.124,E2 -18721.124} C_VEL
LIN {X 0,Y 250.429,Z 402.785,A -85,B 0,C 180,E1 -18724.126,E2 -18724.126} C_VEL
LIN {X 0,Y 249.419,Z 402.908,A -85,B 0,C 180,E1 -18725.474,E2 -18725.474} C_VEL
LIN {X 0,Y 249.379,Z 402.913,A -85,B 0,C 180,E1 -18725.931,E2 -18725.931} C_VEL
LIN {X 0,Y 249.39,Z 402.92,A -85,B 0,C 180,E1 -18729.482,E2 -18729.482} C_VEL
LIN {X 0,Y 249.21,Z 402.941,A -85,B 0,C 180,E1 -18734.703,E2 -18734.703} C_VEL
LIN {X 0,Y 249.144,Z 402.947,A -85,B 0,C 180,E1 -18738.077,E2 -18738.077} C_VEL
LIN {X 0,Y 249.091,Z 402.952,A -85,B 0,C 180,E1 -18741.518,E2 -18741.518} C_VEL
LIN {X 0,Y 249.134,Z 402.952,A -85,B 0,C 180,E1 -18745.482,E2 -18745.482} C_VEL
LIN {X 0,Y 249.076,Z 402.958,A -85,B 0,C 180,E1 -18748.989,E2 -18748.989} C_VEL
LIN {X 0,Y 249.034,Z 402.961,A -85,B 0,C 180,E1 -18752.425,E2 -18752.425} C_VEL
LIN {X 0,Y 249.032,Z 402.961,A -85,B 0,C 180,E1 -18756.345,E2 -18756.345} C_VEL
LIN {X 0,Y 249.009,Z 402.965,A -85,B 0,C 180,E1 -18760.478,E2 -18760.478} C_VEL
LIN {X 0,Y 249.01,Z 402.968,A -85,B 0,C 180,E1 -18764.878,E2 -18764.878} C_VEL
LIN {X 0,Y 249.021,Z 402.967,A -85,B 0,C 180,E1 -18767.363,E2 -18767.363} C_VEL
LIN {X 0,Y 249.04,Z 402.968,A -85,B 0,C 180,E1 -18771.363,E2 -18771.363} C_VEL
LIN {X 0,Y 251.05,Z 411.174,A -85,B 0,C 180,E1 -18775.059,E2 -18775.059} C_VEL
LIN {X 0,Y 252.23,Z 416.067,A -85,B 0,C 180,E1 -18777.079,E2 -18777.079} C_VEL
LIN {X 0,Y 259.677,Z 432.709,A -85,B 0,C 180,E1 -18778.659,E2 -18778.659} C_VEL
LIN {X 0,Y 263.41,Z 442.156,A -85,B 0,C 180,E1 -18779.443,E2 -18779.443} C_VEL
LIN {X 0,Y 266.789,Z 463.744,A -85,B 0,C 180,E1 -18780.523,E2 -18780.523} C_VEL
LIN {X 0,Y 265.677,Z 502.659,A -85,B 0,C 180,E1 -18781.565,E2 -18781.565} C_VEL
LIN {X 0,Y 264.739,Z 525.527,A -85,B 0,C 180,E1 -18782.21,E2 -18782.21} C_VEL
LIN {X 0,Y 263.552,Z 539.056,A -85,B 0,C 180,E1 -18782.881,E2 -18782.881} C_VEL
LIN {X 0,Y 261.946,Z 551.743,A -85,B 0,C 180,E1 -18783.831,E2 -18783.831} C_VEL
LIN {X 0,Y 260.086,Z 563.416,A -85,B 0,C 180,E1 -18785.025,E2 -18785.025} C_VEL
LIN {X 0,Y 258.019,Z 574.693,A -85,B 0,C 180,E1 -18786.524,E2 -18786.524} C_VEL
LIN {X 0,Y 255.774,Z 584.849,A -85,B 0,C 180,E1 -18788.226,E2 -18788.226} C_VEL
LIN {X 0,Y 253.751,Z 594.001,A -85,B 0,C 180,E1 -18790.166,E2 -18790.166} C_VEL
LIN {X 0,Y 252.083,Z 601.567,A -85,B 0,C 180,E1 -18792.14,E2 -18792.14} C_VEL
LIN {X 0,Y 250.298,Z 608.99,A -85,B 0,C 180,E1 -18794.529,E2 -18794.529} C_VEL
LIN {X 0,Y 248.83,Z 614.951,A -85,B 0,C 180,E1 -18796.941,E2 -18796.941} C_VEL
LIN {X 0,Y 247.894,Z 619.666,A -85,B 0,C 180,E1 -18799.38,E2 -18799.38} C_VEL
LIN {X 0,Y 247.269,Z 623.27,A -85,B 0,C 180,E1 -18801.83,E2 -18801.83} C_VEL
LIN {X 0,Y 247.01,Z 625.128,A -85,B 0,C 180,E1 -18803.465,E2 -18803.465} C_VEL
LIN {X 0,Y 246.85,Z 627.519,A -85,B 0,C 180,E1 -18806.735,E2 -18806.735} C_VEL
LIN {X 0,Y 246.897,Z 628.128,A -85,B 0,C 180,E1 -18808.369,E2 -18808.369} C_VEL
LIN {X 0,Y 246.935,Z 628.341,A -85,B 0,C 180,E1 -18810,E2 -18810} C_VEL
LIN {X 0,Y 246.897,Z 628.119,A -85,B 0,C 180,E1 -18811.631,E2 -18811.631} C_VEL
LIN {X 0,Y 246.851,Z 627.504,A -85,B 0,C 180,E1 -18813.264,E2 -18813.264} C_VEL
LIN {X 0,Y 246.882,Z 626.502,A -85,B 0,C 180,E1 -18814.899,E2 -18814.899} C_VEL
LIN {X 0,Y 247.009,Z 625.098,A -85,B 0,C 180,E1 -18816.535,E2 -18816.535} C_VEL
LIN {X 0,Y 247.457,Z 622.154,A -85,B 0,C 180,E1 -18818.986,E2 -18818.986} C_VEL
LIN {X 0,Y 248.175,Z 618.171,A -85,B 0,C 180,E1 -18821.433,E2 -18821.433} C_VEL
LIN {X 0,Y 249.492,Z 612.051,A -85,B 0,C 180,E1 -18824.269,E2 -18824.269} C_VEL
LIN {X 0,Y 251.197,Z 605.373,A -85,B 0,C 180,E1 -18826.665,E2 -18826.665} C_VEL
LIN {X 0,Y 253.135,Z 596.963,A -85,B 0,C 180,E1 -18829.074,E2 -18829.074} C_VEL
LIN {X 0,Y 254.922,Z 588.585,A -85,B 0,C 180,E1 -18831.002,E2 -18831.002} C_VEL
LIN {X 0,Y 257.208,Z 578.088,A -85,B 0,C 180,E1 -18832.915,E2 -18832.915} C_VEL
